u32gTotalDistanceRawValue := TO_UDINT((u32gTotalDistance.Value - u32gTotalDistance.AppScalingOffset) * u32gTotalDistance.AppScalingDivisor / u32gTotalDistance.AppScalingMultiplier);

                  
END_GET
END_PROPERTY

PROPERTY i32gDistanceTraveledMeasureMastToolValue : DINT
GET
                    IF i32gDistanceTraveledMeasureMast.ToolScalingDivisor = 0 OR i32gDistanceTraveledMeasureMast.AppScalingMultiplier = 0 THEN
	_MatchLog^.Error("Get i32gDistanceTraveledMeasureMastToolValue", "Division by Zero!");
	RETURN;
END_IF

i32gDistanceTraveledMeasureMastToolValue := TO_DINT(((i32gDistanceTraveledMeasureMast.Value - i32gDistanceTraveledMeasureMast.AppScalingOffset) * i32gDistanceTraveledMeasureMast.AppScalingDivisor / i32gDistanceTraveledMeasureMast.AppScalingMultiplier * i32gDistanceTraveledMeasureMast.ToolScalingMultiplier / i32gDistanceTraveledMeasureMast.ToolScalingDivisor) + i32gDistanceTraveledMeasureMast.ToolScalingOffset);

                  
END_GET
END_PROPERTY

PROPERTY u32gTotalDistanceToolValue : UDINT
GET
                    IF u32gTotalDistance.ToolScalingDivisor = 0 OR u32gTotalDistance.AppScalingMultiplier = 0 THEN
	_MatchLog^.Error("Get u32gTotalDistanceToolValue", "Division by Zero!");
	RETURN;
END_IF

u32gTotalDistanceToolValue := TO_UDINT(((u32gTotalDistance.Value - u32gTotalDistance.AppScalingOffset) * u32gTotalDistance.AppScalingDivisor / u32gTotalDistance.AppScalingMultiplier * u32gTotalDistance.ToolScalingMultiplier / u32gTotalDistance.ToolScalingDivisor) + u32gTotalDistance.ToolScalingOffset);

                  
END_GET
END_PROPERTY

METHOD InitializeCanSignals
                  i32gDistanceTraveledMeasureMast.AppScalingDivisor :=1;
i32gDistanceTraveledMeasureMast.AppScalingMultiplier :=1;
i32gDistanceTraveledMeasureMast.AppScalingOffset :=0;
i32gDistanceTraveledMeasureMast.AppUnit :="";
i32gDistanceTraveledMeasureMast.CanDefault :=0;
i32gDistanceTraveledMeasureMast.CanInit :=0;
i32gDistanceTraveledMeasureMast.CanMax :=VBasic.LibConst.I32_MAX;
i32gDistanceTraveledMeasureMast.CanMin :=VBasic.LibConst.32_MIN;
i32gDistanceTraveledMeasureMast.CanUnit :="";
i32gDistanceTraveledMeasureMast.Description :="new signal";
i32gDistanceTraveledMeasureMast.ErrorReaction := eErrorReaction.ERSIG_DFLT;
i32gDistanceTraveledMeasureMast.ReceiverAdress :=1;
i32gDistanceTraveledMeasureMast.ToolScalingDivisor :=1;
i32gDistanceTraveledMeasureMast.ToolScalingMultiplier :=1;
i32gDistanceTraveledMeasureMast.ToolScalingOffset :=0;
i32gDistanceTraveledMeasureMast.ToolUnit :="";

u32gTotalDistance.AppScalingDivisor :=1;
u32gTotalDistance.AppScalingMultiplier :=1;
u32gTotalDistance.AppScalingOffset :=0;
u32gTotalDistance.AppUnit :="";
u32gTotalDistance.CanDefault :=0;
u32gTotalDistance.CanInit :=0;
u32gTotalDistance.CanMax :=VBasic.LibConst.U32_MAX;
u32gTotalDistance.CanMin :=VBasic.LibConst.U32_MIN;
u32gTotalDistance.CanUnit :="";
u32gTotalDistance.Description :="new signal";
u32gTotalDistance.ErrorReaction := eErrorReaction.ERSIG_DFLT;
u32gTotalDistance.ReceiverAdress :=1;
u32gTotalDistance.ToolScalingDivisor :=1;
u32gTotalDistance.ToolScalingMultiplier :=1;
u32gTotalDistance.ToolScalingOffset :=0;
u32gTotalDistance.ToolUnit :="";


                
END_METHOD
END_FUNCTION_BLOCK

FUNCTION_BLOCK Msg13C0SendToEvision7MessageClass EXTENDS CanReceiveMessageClass
  VAR_INPUT
    u8gReductionPumpRail : UInt8CanSignalClass;
    u8gPourcentCycleBrake : UInt8CanSignalClass;
    u8gPourcentCycle2ndParkBrake : UInt8CanSignalClass;
    bogSecondParkBrakeActive : BoolCanSignalClass;
    boStatFront2eParkTrainBrakeTest : BoolCanSignalClass;
    boStatBack2eParkTrainBrakeTest : BoolCanSignalClass;
    boAutorizeRazController : BoolCanSignalClass;
    boVoltageDcConverterFault : BoolCanSignalClass;
    boBatteryLowLevel : BoolCanSignalClass;
    boBattErrorCode1 : BoolCanSignalClass;
    boActiveFaultRazDmc : BoolCanSignalClass;
    i16Motor_Rpm : Int16CanSignalClass;
    i8Controller_Temp : Int8CanSignalClass;
    i8Motor_Temp : Int8CanSignalClass;
    Counter : UInt32CanSignalClass;
  END_VAR

            
          

METHOD SetData
  VAR_INPUT
    CanMsgPointer : POINTER TO CanMessageClass;
  END_VAR
                  IF IsValidPointer(canMsgPointer,'SetData') THEN
	SUPER^.SetData(CanMsgPointer);
	//Set the new data
	u8gReductionPumpRail.Value := canMsgPointer^.GetUint8(0);
	u8gPourcentCycleBrake.Value := canMsgPointer^.GetUint8(8);
	u8gPourcentCycle2ndParkBrake.Value := canMsgPointer^.GetUint8(16);
	bogSecondParkBrakeActive.Value := canMsgPointer^.GetBoolOnBit(24);
	boStatFront2eParkTrainBrakeTest.Value := canMsgPointer^.GetBoolOnBit(25);
	boStatBack2eParkTrainBrakeTest.Value := canMsgPointer^.GetBoolOnBit(26);
	boAutorizeRazController.Value := canMsgPointer^.GetBoolOnBit(27);
	boVoltageDcConverterFault.Value := canMsgPointer^.GetBoolOnBit(28);
	boBatteryLowLevel.Value := canMsgPointer^.GetBoolOnBit(29);
	boBattErrorCode1.Value := canMsgPointer^.GetBoolOnBit(30);
	boActiveFaultRazDmc.Value := canMsgPointer^.GetBoolOnBit(31);
	i16Motor_Rpm.Value := canMsgPointer^.GetInt16(32);
	i8Controller_Temp.Value := canMsgPointer^.GetInt8(48);
	i8Motor_Temp.Value := canMsgPointer^.GetInt8(56);
	//And increase the counter
	Counter.Value := CanMsgPointer^.Counter.Value;
END_IF

                
END_METHOD

PROPERTY u8gReductionPumpRailRawValue : USINT
GET
                    IF u8gReductionPumpRail.AppScalingMultiplier = 0 THEN
	_MatchLog^.Error("Get u8gReductionPumpRailRawValue", "Division by Zero!");
	RETURN;
End_IF

u8gReductionPumpRailRawValue := TO_USINT((u8gReductionPumpRail.Value - u8gReductionPumpRail.AppScalingOffset) * u8gReductionPumpRail.AppScalingDivisor / u8gReductionPumpRail.AppScalingMultiplier);

                  
END_GET
END_PROPERTY

PROPERTY u8gPourcentCycleBrakeRawValue : USINT
GET
                    IF u8gPourcentCycleBrake.AppScalingMultiplier = 0 THEN
	_MatchLog^.Error("Get u8gPourcentCycleBrakeRawValue", "Division by Zero!");
	RETURN;
End_IF

u8gPourcentCycleBrakeRawValue := TO_USINT((u8gPourcentCycleBrake.Value - u8gPourcentCycleBrake.AppScalingOffset) * u8gPourcentCycleBrake.AppScalingDivisor / u8gPourcentCycleBrake.AppScalingMultiplier);

                  
END_GET
END_PROPERTY

PROPERTY u8gPourcentCycle2ndParkBrakeRawValue : USINT
GET
                    IF u8gPourcentCycle2ndParkBrake.AppScalingMultiplier = 0 THEN
	_MatchLog^.Error("Get u8gPourcentCycle2ndParkBrakeRawValue", "Division by Zero!");
	RETURN;
End_IF

u8gPourcentCycle2ndParkBrakeRawValue := TO_USINT((u8gPourcentCycle2ndParkBrake.Value - u8gPourcentCycle2ndParkBrake.AppScalingOffset) * u8gPourcentCycle2ndParkBrake.AppScalingDivisor / u8gPourcentCycle2ndParkBrake.AppScalingMultiplier);

                  
END_GET
END_PROPERTY

PROPERTY bogSecondParkBrakeActiveRawValue : BOOL
GET
                    bogSecondParkBrakeActiveRawValue := bogSecondParkBrakeActive.Value;

                  
END_GET
END_PROPERTY

PROPERTY boStatFront2eParkTrainBrakeTestRawValue : BOOL
GET
                    boStatFront2eParkTrainBrakeTestRawValue := boStatFront2eParkTrainBrakeTest.Value;

                  
END_GET
END_PROPERTY

PROPERTY boStatBack2eParkTrainBrakeTestRawValue : BOOL
GET
                    boStatBack2eParkTrainBrakeTestRawValue := boStatBack2eParkTrainBrakeTest.Value;

                  
END_GET
END_PROPERTY

PROPERTY boAutorizeRazControllerRawValue : BOOL
GET
                    boAutorizeRazControllerRawValue := boAutorizeRazController.Value;

                  
END_GET
END_PROPERTY

PROPERTY boVoltageDcConverterFaultRawValue : BOOL
GET
                    boVoltageDcConverterFaultRawValue := boVoltageDcConverterFault.Value;

                  
END_GET
END_PROPERTY

PROPERTY boBatteryLowLevelRawValue : BOOL
GET
                    boBatteryLowLevelRawValue := boBatteryLowLevel.Value;

                  
END_GET
END_PROPERTY

PROPERTY boBattErrorCode1RawValue : BOOL
GET
                    boBattErrorCode1RawValue := boBattErrorCode1.Value;

                  
END_GET
END_PROPERTY

PROPERTY boActiveFaultRazDmcRawValue : BOOL
GET
                    boActiveFaultRazDmcRawValue := boActiveFaultRazDmc.Value;

                  
END_GET
END_PROPERTY

PROPERTY i16Motor_RpmRawValue : INT
GET
                    IF i16Motor_Rpm.AppScalingMultiplier = 0 THEN
	_MatchLog^.Error("Get i16Motor_RpmRawValue", "Division by Zero!");
	RETURN;
End_IF

i16Motor_RpmRawValue := TO_INT((i16Motor_Rpm.Value - i16Motor_Rpm.AppScalingOffset) * i16Motor_Rpm.AppScalingDivisor / i16Motor_Rpm.AppScalingMultiplier);

                  
END_GET
END_PROPERTY

PROPERTY i8Controller_TempRawValue : SINT
GET
                    IF i8Controller_Temp.AppScalingMultiplier = 0 THEN
	_MatchLog^.Error("Get i8Controller_TempRawValue", "Division by Zero!");
	RETURN;
End_IF

i8Controller_TempRawValue := TO_SINT((i8Controller_Temp.Value - i8Controller_Temp.AppScalingOffset) * i8Controller_Temp.AppScalingDivisor / i8Controller_Temp.AppScalingMultiplier);

                  
END_GET
END_PROPERTY

PROPERTY i8Motor_TempRawValue : SINT
GET
                    IF i8Motor_Temp.AppScalingMultiplier = 0 THEN
	_MatchLog^.Error("Get i8Motor_TempRawValue", "Division by Zero!");
	RETURN;
End_IF

i8Motor_TempRawValue := TO_SINT((i8Motor_Temp.Value - i8Motor_Temp.AppScalingOffset) * i8Motor_Temp.AppScalingDivisor / i8Motor_Temp.AppScalingMultiplier);

                  
END_GET
END_PROPERTY

PROPERTY u8gReductionPumpRailToolValue : USINT
GET
                    IF u8gReductionPumpRail.ToolScalingDivisor = 0 OR u8gReductionPumpRail.AppScalingMultiplier = 0 THEN
	_MatchLog^.Error("Get u8gReductionPumpRailToolValue", "Division by Zero!");
	RETURN;
END_IF

u8gReductionPumpRailToolValue := TO_USINT(((u8gReductionPumpRail.Value - u8gReductionPumpRail.AppScalingOffset) * u8gReductionPumpRail.AppScalingDivisor / u8gReductionPumpRail.AppScalingMultiplier * u8gReductionPumpRail.ToolScalingMultiplier / u8gReductionPumpRail.ToolScalingDivisor) + u8gReductionPumpRail.ToolScalingOffset);

                  
END_GET
END_PROPERTY

PROPERTY u8gPourcentCycleBrakeToolValue : USINT
GET
                    IF u8gPourcentCycleBrake.ToolScalingDivisor = 0 OR u8gPourcentCycleBrake.AppScalingMultiplier = 0 THEN
	_MatchLog^.Error("Get u8gPourcentCycleBrakeToolValue", "Division by Zero!");
	RETURN;
END_IF

u8gPourcentCycleBrakeToolValue := TO_USINT(((u8gPourcentCycleBrake.Value - u8gPourcentCycleBrake.AppScalingOffset) * u8gPourcentCycleBrake.AppScalingDivisor / u8gPourcentCycleBrake.AppScalingMultiplier * u8gPourcentCycleBrake.ToolScalingMultiplier / u8gPourcentCycleBrake.ToolScalingDivisor) + u8gPourcentCycleBrake.ToolScalingOffset);

                  
END_GET
END_PROPERTY

PROPERTY u8gPourcentCycle2ndParkBrakeToolValue : USINT
GET
                    IF u8gPourcentCycle2ndParkBrake.ToolScalingDivisor = 0 OR u8gPourcentCycle2ndParkBrake.AppScalingMultiplier = 0 THEN
	_MatchLog^.Error("Get u8gPourcentCycle2ndParkBrakeToolValue", "Division by Zero!");
	RETURN;
END_IF

u8gPourcentCycle2ndParkBrakeToolValue := TO_USINT(((u8gPourcentCycle2ndParkBrake.Value - u8gPourcentCycle2ndParkBrake.AppScalingOffset) * u8gPourcentCycle2ndParkBrake.AppScalingDivisor / u8gPourcentCycle2ndParkBrake.AppScalingMultiplier * u8gPourcentCycle2ndParkBrake.ToolScalingMultiplier / u8gPourcentCycle2ndParkBrake.ToolScalingDivisor) + u8gPourcentCycle2ndParkBrake.ToolScalingOffset);

                  
END_GET
END_PROPERTY

PROPERTY bogSecondParkBrakeActiveToolValue : BOOL
GET
                    bogSecondParkBrakeActiveToolValue := bogSecondParkBrakeActive.Value;

                  
END_GET
END_PROPERTY

PROPERTY boStatFront2eParkTrainBrakeTestToolValue : BOOL
GET
                    boStatFront2eParkTrainBrakeTestToolValue := boStatFront2eParkTrainBrakeTest.Value;

                  
END_GET
END_PROPERTY

PROPERTY boStatBack2eParkTrainBrakeTestToolValue : BOOL
GET
                    boStatBack2eParkTrainBrakeTestToolValue := boStatBack2eParkTrainBrakeTest.Value;

                  
END_GET
END_PROPERTY

PROPERTY boAutorizeRazControllerToolValue : BOOL
GET
                    boAutorizeRazControllerToolValue := boAutorizeRazController.Value;

                  
END_GET
END_PROPERTY

PROPERTY boVoltageDcConverterFaultToolValue : BOOL
GET
                    boVoltageDcConverterFaultToolValue := boVoltageDcConverterFault.Value;

                  
END_GET
END_PROPERTY

PROPERTY boBatteryLowLevelToolValue : BOOL
GET
                    boBatteryLowLevelToolValue := boBatteryLowLevel.Value;

                  
END_GET
END_PROPERTY

PROPERTY boBattErrorCode1ToolValue : BOOL
GET
                    boBattErrorCode1ToolValue := boBattErrorCode1.Value;

                  
END_GET
END_PROPERTY

PROPERTY boActiveFaultRazDmcToolValue : BOOL
GET
                    boActiveFaultRazDmcToolValue := boActiveFaultRazDmc.Value;

                  
END_GET
END_PROPERTY

PROPERTY i16Motor_RpmToolValue : INT
GET
                    IF i16Motor_Rpm.ToolScalingDivisor = 0 OR i16Motor_Rpm.AppScalingMultiplier = 0 THEN
	_MatchLog^.Error("Get i16Motor_RpmToolValue", "Division by Zero!");
	RETURN;
END_IF

i16Motor_RpmToolValue := TO_INT(((i16Motor_Rpm.Value - i16Motor_Rpm.AppScalingOffset) * i16Motor_Rpm.AppScalingDivisor / i16Motor_Rpm.AppScalingMultiplier * i16Motor_Rpm.ToolScalingMultiplier / i16Motor_Rpm.ToolScalingDivisor) + i16Motor_Rpm.ToolScalingOffset);

                  
END_GET
END_PROPERTY

PROPERTY i8Controller_TempToolValue : SINT
GET
                    IF i8Controller_Temp.ToolScalingDivisor = 0 OR i8Controller_Temp.AppScalingMultiplier = 0 THEN
	_MatchLog^.Error("Get i8Controller_TempToolValue", "Division by Zero!");
	RETURN;
END_IF

i8Controller_TempToolValue := TO_SINT(((i8Controller_Temp.Value - i8Controller_Temp.AppScalingOffset) * i8Controller_Temp.AppScalingDivisor / i8Controller_Temp.AppScalingMultiplier * i8Controller_Temp.ToolScalingMultiplier / i8Controller_Temp.ToolScalingDivisor) + i8Controller_Temp.ToolScalingOffset);

                  
END_GET
END_PROPERTY

PROPERTY i8Motor_TempToolValue : SINT
GET
                    IF i8Motor_Temp.ToolScalingDivisor = 0 OR i8Motor_Temp.AppScalingMultiplier = 0 THEN
	_MatchLog^.Error("Get i8Motor_TempToolValue", "Division by Zero!");
	RETURN;
END_IF

i8Motor_TempToolValue := TO_SINT(((i8Motor_Temp.Value - i8Motor_Temp.AppScalingOffset) * i8Motor_Temp.AppScalingDivisor / i8Motor_Temp.AppScalingMultiplier * i8Motor_Temp.ToolScalingMultiplier / i8Motor_Temp.ToolScalingDivisor) + i8Motor_Temp.ToolScalingOffset);

                  
END_GET
END_PROPERTY

METHOD InitializeCanSignals
                  u8gReductionPumpRail.AppScalingDivisor :=1;
u8gReductionPumpRail.AppScalingMultiplier :=1;
u8gReductionPumpRail.AppScalingOffset :=0;
u8gReductionPumpRail.AppUnit :="";
u8gReductionPumpRail.CanDefault :=0;
u8gReductionPumpRail.CanInit :=0;
u8gReductionPumpRail.CanMax :=VBasic.LibConst.U8_MAX;
u8gReductionPumpRail.CanMin :=VBasic.LibConst.U8_MIN;
u8gReductionPumpRail.CanUnit :="";
u8gReductionPumpRail.Description :="new signal";
u8gReductionPumpRail.ErrorReaction := eErrorReaction.ERSIG_DFLT;
u8gReductionPumpRail.ReceiverAdress :=1;
u8gReductionPumpRail.ToolScalingDivisor :=1;
u8gReductionPumpRail.ToolScalingMultiplier :=1;
u8gReductionPumpRail.ToolScalingOffset :=0;
u8gReductionPumpRail.ToolUnit :="";

u8gPourcentCycleBrake.AppScalingDivisor :=1;
u8gPourcentCycleBrake.AppScalingMultiplier :=1;
u8gPourcentCycleBrake.AppScalingOffset :=0;
u8gPourcentCycleBrake.AppUnit :="";
u8gPourcentCycleBrake.CanDefault :=0;
u8gPourcentCycleBrake.CanInit :=0;
u8gPourcentCycleBrake.CanMax :=VBasic.LibConst.U8_MAX;
u8gPourcentCycleBrake.CanMin :=VBasic.LibConst.U8_MIN;
u8gPourcentCycleBrake.CanUnit :="";
u8gPourcentCycleBrake.Description :="new signal";
u8gPourcentCycleBrake.ErrorReaction := eErrorReaction.ERSIG_DFLT;
u8gPourcentCycleBrake.ReceiverAdress :=1;
u8gPourcentCycleBrake.ToolScalingDivisor :=1;
u8gPourcentCycleBrake.ToolScalingMultiplier :=1;
u8gPourcentCycleBrake.ToolScalingOffset :=0;
u8gPourcentCycleBrake.ToolUnit :="";

u8gPourcentCycle2ndParkBrake.AppScalingDivisor :=1;
u8gPourcentCycle2ndParkBrake.AppScalingMultiplier :=1;
u8gPourcentCycle2ndParkBrake.AppScalingOffset :=0;
u8gPourcentCycle2ndParkBrake.AppUnit :="";
u8gPourcentCycle2ndParkBrake.CanDefault :=0;
u8gPourcentCycle2ndParkBrake.CanInit :=0;
u8gPourcentCycle2ndParkBrake.CanMax :=VBasic.LibConst.U8_MAX;
u8gPourcentCycle2ndParkBrake.CanMin :=VBasic.LibConst.U8_MIN;
u8gPourcentCycle2ndParkBrake.CanUnit :="";
u8gPourcentCycle2ndParkBrake.Description :="Envoie du pourcentage du nombre de cycle de freins";
u8gPourcentCycle2ndParkBrake.ErrorReaction := eErrorReaction.ERSIG_DFLT;
u8gPourcentCycle2ndParkBrake.ReceiverAdress :=1;
u8gPourcentCycle2ndParkBrake.ToolScalingDivisor :=1;
u8gPourcentCycle2ndParkBrake.ToolScalingMultiplier :=1;
u8gPourcentCycle2ndParkBrake.ToolScalingOffset :=0;
u8gPourcentCycle2ndParkBrake.ToolUnit :="";

bogSecondParkBrakeActive.AppScalingDivisor :=1;
bogSecondParkBrakeActive.AppScalingMultiplier :=1;
bogSecondParkBrakeActive.AppScalingOffset :=0;
bogSecondParkBrakeActive.AppUnit :="";
bogSecondParkBrakeActive.CanDefault :=0;
bogSecondParkBrakeActive.CanInit :=0;
bogSecondParkBrakeActive.CanMax :=1;
bogSecondParkBrakeActive.CanMin :=0;
bogSecondParkBrakeActive.CanUnit :="";
bogSecondParkBrakeActive.Description :="Option active";
bogSecondParkBrakeActive.ErrorReaction := eErrorReaction.ERSIG_DFLT;
bogSecondParkBrakeActive.ReceiverAdress :=1;
bogSecondParkBrakeActive.ToolScalingDivisor :=1;
bogSecondParkBrakeActive.ToolScalingMultiplier :=1;
bogSecondParkBrakeActive.ToolScalingOffset :=0;
bogSecondParkBrakeActive.ToolUnit :="";

boStatFront2eParkTrainBrakeTest.AppScalingDivisor :=1;
boStatFront2eParkTrainBrakeTest.AppScalingMultiplier :=1;
boStatFront2eParkTrainBrakeTest.AppScalingOffset :=0;
boStatFront2eParkTrainBrakeTest.AppUnit :="";
boStatFront2eParkTrainBrakeTest.CanDefault :=0;
boStatFront2eParkTrainBrakeTest.CanInit :=0;
boStatFront2eParkTrainBrakeTest.CanMax :=1;
boStatFront2eParkTrainBrakeTest.CanMin :=0;
boStatFront2eParkTrainBrakeTest.CanUnit :="";
boStatFront2eParkTrainBrakeTest.Description :="Validation du test frein sur le 2nd frein de oscillant";
boStatFront2eParkTrainBrakeTest.ErrorReaction := eErrorReaction.ERSIG_DFLT;
boStatFront2eParkTrainBrakeTest.ReceiverAdress :=1;
boStatFront2eParkTrainBrakeTest.ToolScalingDivisor :=1;
boStatFront2eParkTrainBrakeTest.ToolScalingMultiplier :=1;
boStatFront2eParkTrainBrakeTest.ToolScalingOffset :=0;
boStatFront2eParkTrainBrakeTest.ToolUnit :="";

boStatBack2eParkTrainBrakeTest.AppScalingDivisor :=1;
boStatBack2eParkTrainBrakeTest.AppScalingMultiplier :=1;
boStatBack2eParkTrainBrakeTest.AppScalingOffset :=0;
boStatBack2eParkTrainBrakeTest.AppUnit :="";
boStatBack2eParkTrainBrakeTest.CanDefault :=0;
boStatBack2eParkTrainBrakeTest.CanInit :=0;
boStatBack2eParkTrainBrakeTest.CanMax :=1;
boStatBack2eParkTrainBrakeTest.CanMin :=0;
boStatBack2eParkTrainBrakeTest.CanUnit :="";
boStatBack2eParkTrainBrakeTest.Description :="Validation du test frein sur le 2nd frein du fixe";
boStatBack2eParkTrainBrakeTest.ErrorReaction := eErrorReaction.ERSIG_DFLT;
boStatBack2eParkTrainBrakeTest.ReceiverAdress :=1;
boStatBack2eParkTrainBrakeTest.ToolScalingDivisor :=1;
boStatBack2eParkTrainBrakeTest.ToolScalingMultiplier :=1;
boStatBack2eParkTrainBrakeTest.ToolScalingOffset :=0;
boStatBack2eParkTrainBrakeTest.ToolUnit :="";

boAutorizeRazController.AppScalingDivisor :=1;
boAutorizeRazController.AppScalingMultiplier :=1;
boAutorizeRazController.AppScalingOffset :=0;
boAutorizeRazController.AppUnit :="";
boAutorizeRazController.CanDefault :=0;
boAutorizeRazController.CanInit :=0;
boAutorizeRazController.CanMax :=1;
boAutorizeRazController.CanMin :=0;
boAutorizeRazController.CanUnit :="";
boAutorizeRazController.Description :="new signal";
boAutorizeRazController.ErrorReaction := eErrorReaction.ERSIG_DFLT;
boAutorizeRazController.ReceiverAdress :=1;
boAutorizeRazController.ToolScalingDivisor :=1;
boAutorizeRazController.ToolScalingMultiplier :=1;
boAutorizeRazController.ToolScalingOffset :=0;
boAutorizeRazController.ToolUnit :="";

boVoltageDcConverterFault.AppScalingDivisor :=1;
boVoltageDcConverterFault.AppScalingMultiplier :=1;
boVoltageDcConverterFault.AppScalingOffset :=0;
boVoltageDcConverterFault.AppUnit :="";
boVoltageDcConverterFault.CanDefault :=0;
boVoltageDcConverterFault.CanInit :=0;
boVoltageDcConverterFault.CanMax :=1;
boVoltageDcConverterFault.CanMin :=0;
boVoltageDcConverterFault.CanUnit :="";
boVoltageDcConverterFault.Description :="new signal";
boVoltageDcConverterFault.ErrorReaction := eErrorReaction.ERSIG_DFLT;
boVoltageDcConverterFault.ReceiverAdress :=1;
boVoltageDcConverterFault.ToolScalingDivisor :=1;
boVoltageDcConverterFault.ToolScalingMultiplier :=1;
boVoltageDcConverterFault.ToolScalingOffset :=0;
boVoltageDcConverterFault.ToolUnit :="";

boBatteryLowLevel.AppScalingDivisor :=1;
boBatteryLowLevel.AppScalingMultiplier :=1;
boBatteryLowLevel.AppScalingOffset :=0;
boBatteryLowLevel.AppUnit :="";
boBatteryLowLevel.CanDefault :=0;
boBatteryLowLevel.CanInit :=0;
boBatteryLowLevel.CanMax :=1;
boBatteryLowLevel.CanMin :=0;
boBatteryLowLevel.CanUnit :="";
boBatteryLowLevel.Description :="new signal";
boBatteryLowLevel.ErrorReaction := eErrorReaction.ERSIG_DFLT;
boBatteryLowLevel.ReceiverAdress :=1;
boBatteryLowLevel.ToolScalingDivisor :=1;
boBatteryLowLevel.ToolScalingMultiplier :=1;
boBatteryLowLevel.ToolScalingOffset :=0;
boBatteryLowLevel.ToolUnit :="";

boBattErrorCode1.AppScalingDivisor :=1;
boBattErrorCode1.AppScalingMultiplier :=1;
boBattErrorCode1.AppScalingOffset :=0;
boBattErrorCode1.AppUnit :="";
boBattErrorCode1.CanDefault :=0;
boBattErrorCode1.CanInit :=0;
boBattErrorCode1.CanMax :=1;
boBattErrorCode1.CanMin :=0;
boBattErrorCode1.CanUnit :="";
boBattErrorCode1.Description :="new signal";
boBattErrorCode1.ErrorReaction := eErrorReaction.ERSIG_DFLT;
boBattErrorCode1.ReceiverAdress :=1;
boBattErrorCode1.ToolScalingDivisor :=1;
boBattErrorCode1.ToolScalingMultiplier :=1;
boBattErrorCode1.ToolScalingOffset :=0;
boBattErrorCode1.ToolUnit :="";

boActiveFaultRazDmc.AppScalingDivisor :=1;
boActiveFaultRazDmc.AppScalingMultiplier :=1;
boActiveFaultRazDmc.AppScalingOffset :=0;
boActiveFaultRazDmc.AppUnit :="";
boActiveFaultRazDmc.CanDefault :=0;
boActiveFaultRazDmc.CanInit :=0;
boActiveFaultRazDmc.CanMax :=1;
boActiveFaultRazDmc.CanMin :=0;
boActiveFaultRazDmc.CanUnit :="";
boActiveFaultRazDmc.Description :="new signal";
boActiveFaultRazDmc.ErrorReaction := eErrorReaction.ERSIG_DFLT;
boActiveFaultRazDmc.ReceiverAdress :=1;
boActiveFaultRazDmc.ToolScalingDivisor :=1;
boActiveFaultRazDmc.ToolScalingMultiplier :=1;
boActiveFaultRazDmc.ToolScalingOffset :=0;
boActiveFaultRazDmc.ToolUnit :="";

i16Motor_Rpm.AppScalingDivisor :=1;
i16Motor_Rpm.AppScalingMultiplier :=1;
i16Motor_Rpm.AppScalingOffset :=0;
i16Motor_Rpm.AppUnit :="";
i16Motor_Rpm.CanDefault :=0;
i16Motor_Rpm.CanInit :=0;
i16Motor_Rpm.CanMax :=VBasic.LibConst.I16_MAX;
i16Motor_Rpm.CanMin :=VBasic.LibConst.I16_MIN;
i16Motor_Rpm.CanUnit :="";
i16Motor_Rpm.Description :="new signal";
i16Motor_Rpm.ErrorReaction := eErrorReaction.ERSIG_DFLT;
i16Motor_Rpm.ReceiverAdress :=1;
i16Motor_Rpm.ToolScalingDivisor :=1;
i16Motor_Rpm.ToolScalingMultiplier :=1;
i16Motor_Rpm.ToolScalingOffset :=0;
i16Motor_Rpm.ToolUnit :="";

i8Controller_Temp.AppScalingDivisor :=1;
i8Controller_Temp.AppScalingMultiplier :=1;
i8Controller_Temp.AppScalingOffset :=0;
i8Controller_Temp.AppUnit :="";
i8Controller_Temp.CanDefault :=0;
i8Controller_Temp.CanInit :=0;
i8Controller_Temp.CanMax :=VBasic.LibConst.I8_MAX;
i8Controller_Temp.CanMin :=VBasic.LibConst.I8_MIN;
i8Controller_Temp.CanUnit :="";
i8Controller_Temp.Description :="new signal";
i8Controller_Temp.ErrorReaction := eErrorReaction.ERSIG_DFLT;
i8Controller_Temp.ReceiverAdress :=1;
i8Controller_Temp.ToolScalingDivisor :=1;
i8Controller_Temp.ToolScalingMultiplier :=1;
i8Controller_Temp.ToolScalingOffset :=0;
i8Controller_Temp.ToolUnit :="";

i8Motor_Temp.AppScalingDivisor :=1;
i8Motor_Temp.AppScalingMultiplier :=1;
i8Motor_Temp.AppScalingOffset :=0;
i8Motor_Temp.AppUnit :="";
i8Motor_Temp.CanDefault :=0;
i8Motor_Temp.CanInit :=0;
i8Motor_Temp.CanMax :=VBasic.LibConst.I8_MAX;
i8Motor_Temp.CanMin :=VBasic.LibConst.I8_MIN;
i8Motor_Temp.CanUnit :="";
i8Motor_Temp.Description :="new signal";
i8Motor_Temp.ErrorReaction := eErrorReaction.ERSIG_DFLT;
i8Motor_Temp.ReceiverAdress :=1;
i8Motor_Temp.ToolScalingDivisor :=1;
i8Motor_Temp.ToolScalingMultiplier :=1;
i8Motor_Temp.ToolScalingOffset :=0;
i8Motor_Temp.ToolUnit :="";


                
END_METHOD
END_FUNCTION_BLOCK

FUNCTION_BLOCK Msg14C0SendToEvision7MessageClass EXTENDS CanReceiveMessageClass
  VAR_INPUT
    i16Ibatt_ist : Int16CanSignalClass;
    u16Vbatt_ist : UInt16CanSignalClass;
    u8Batt_Soc : UInt8CanSignalClass;
    boAddParkBrakeActive : BoolCanSignalClass;
    boPreventLimitSpeedExceeding : BoolCanSignalClass;
    Counter : UInt32CanSignalClass;
  END_VAR

            
          

METHOD SetData
  VAR_INPUT
    CanMsgPointer : POINTER TO CanMessageClass;
  END_VAR
                  IF IsValidPointer(canMsgPointer,'SetData') THEN
	SUPER^.SetData(CanMsgPointer);
	//Set the new data
	i16Ibatt_ist.Value := canMsgPointer^.GetInt16(0);
	u16Vbatt_ist.Value := canMsgPointer^.GetUint16(16);
	u8Batt_Soc.Value := canMsgPointer^.GetUint8(32);
	boAddParkBrakeActive.Value := canMsgPointer^.GetBoolOnBit(56);
	boPreventLimitSpeedExceeding.Value := canMsgPointer^.GetBoolOnBit(57);
	//And increase the counter
	Counter.Value := CanMsgPointer^.Counter.Value;
END_IF

                
END_METHOD

PROPERTY i16Ibatt_istRawValue : INT
GET
                    IF i16Ibatt_ist.AppScalingMultiplier = 0 THEN
	_MatchLog^.Error("Get i16Ibatt_istRawValue", "Division by Zero!");
	RETURN;
End_IF

i16Ibatt_istRawValue := TO_INT((i16Ibatt_ist.Value - i16Ibatt_ist.AppScalingOffset) * i16Ibatt_ist.AppScalingDivisor / i16Ibatt_ist.AppScalingMultiplier);

                  
END_GET
END_PROPERTY

PROPERTY u16Vbatt_istRawValue : UINT
GET
                    IF u16Vbatt_ist.AppScalingMultiplier = 0 THEN
	_MatchLog^.Error("Get u16Vbatt_istRawValue", "Division by Zero!");
	RETURN;
End_IF

u16Vbatt_istRawValue := TO_UINT((u16Vbatt_ist.Value - u16Vbatt_ist.AppScalingOffset) * u16Vbatt_ist.AppScalingDivisor / u16Vbatt_ist.AppScalingMultiplier);

                  
END_GET
END_PROPERTY

PROPERTY u8Batt_SocRawValue : USINT
GET
                    IF u8Batt_Soc.AppScalingMultiplier = 0 THEN
	_MatchLog^.Error("Get u8Batt_SocRawValue", "Division by Zero!");
	RETURN;
End_IF

u8Batt_SocRawValue := TO_USINT((u8Batt_Soc.Value - u8Batt_Soc.AppScalingOffset) * u8Batt_Soc.AppScalingDivisor / u8Batt_Soc.AppScalingMultiplier);

                  
END_GET
END_PROPERTY

PROPERTY boAddParkBrakeActiveRawValue : BOOL
GET
                    boAddParkBrakeActiveRawValue := boAddParkBrakeActive.Value;

                  
END_GET
END_PROPERTY

PROPERTY boPreventLimitSpeedExceedingRawValue : BOOL
GET
                    boPreventLimitSpeedExceedingRawValue := boPreventLimitSpeedExceeding.Value;

                  
END_GET
END_PROPERTY

PROPERTY i16Ibatt_istToolValue : INT
GET
                    IF i16Ibatt_ist.ToolScalingDivisor = 0 OR i16Ibatt_ist.AppScalingMultiplier = 0 THEN
	_MatchLog^.Error("Get i16Ibatt_istToolValue", "Division by Zero!");
	RETURN;
END_IF

i16Ibatt_istToolValue := TO_INT(((i16Ibatt_ist.Value - i16Ibatt_ist.AppScalingOffset) * i16Ibatt_ist.AppScalingDivisor / i16Ibatt_ist.AppScalingMultiplier * i16Ibatt_ist.ToolScalingMultiplier / i16Ibatt_ist.ToolScalingDivisor) + i16Ibatt_ist.ToolScalingOffset);

                  
END_GET
END_PROPERTY

PROPERTY u16Vbatt_istToolValue : UINT
GET
                    IF u16Vbatt_ist.ToolScalingDivisor = 0 OR u16Vbatt_ist.AppScalingMultiplier = 0 THEN
	_MatchLog^.Error("Get u16Vbatt_istToolValue", "Division by Zero!");
	RETURN;
END_IF

u16Vbatt_istToolValue := TO_UINT(((u16Vbatt_ist.Value - u16Vbatt_ist.AppScalingOffset) * u16Vbatt_ist.AppScalingDivisor / u16Vbatt_ist.AppScalingMultiplier * u16Vbatt_ist.ToolScalingMultiplier / u16Vbatt_ist.ToolScalingDivisor) + u16Vbatt_ist.ToolScalingOffset);

                  
END_GET
END_PROPERTY

PROPERTY u8Batt_SocToolValue : USINT
GET
                    IF u8Batt_Soc.ToolScalingDivisor = 0 OR u8Batt_Soc.AppScalingMultiplier = 0 THEN
	_MatchLog^.Error("Get u8Batt_SocToolValue", "Division by Zero!");
	RETURN;
END_IF

u8Batt_SocToolValue := TO_USINT(((u8Batt_Soc.Value - u8Batt_Soc.AppScalingOffset) * u8Batt_Soc.AppScalingDivisor / u8Batt_Soc.AppScalingMultiplier * u8Batt_Soc.ToolScalingMultiplier / u8Batt_Soc.ToolScalingDivisor) + u8Batt_Soc.ToolScalingOffset);

                  
END_GET
END_PROPERTY

PROPERTY boAddParkBrakeActiveToolValue : BOOL
GET
                    boAddParkBrakeActiveToolValue := boAddParkBrakeActive.Value;

                  
END_GET
END_PROPERTY

PROPERTY boPreventLimitSpeedExceedingToolValue : BOOL
GET
                    boPreventLimitSpeedExceedingToolValue := boPreventLimitSpeedExceeding.Value;

                  
END_GET
END_PROPERTY

METHOD InitializeCanSignals
                  i16Ibatt_ist.AppScalingDivisor :=1;
i16Ibatt_ist.AppScalingMultiplier :=1;
i16Ibatt_ist.AppScalingOffset :=0;
i16Ibatt_ist.AppUnit :="";
i16Ibatt_ist.CanDefault :=0;
i16Ibatt_ist.CanInit :=0;
i16Ibatt_ist.CanMax :=VBasic.LibConst.I16_MAX;
i16Ibatt_ist.CanMin :=VBasic.LibConst.I16_MIN;
i16Ibatt_ist.CanUnit :="";
i16Ibatt_ist.Description :="new signal";
i16Ibatt_ist.ErrorReaction := eErrorReaction.ERSIG_DFLT;
i16Ibatt_ist.ReceiverAdress :=1;
i16Ibatt_ist.ToolScalingDivisor :=1;
i16Ibatt_ist.ToolScalingMultiplier :=1;
i16Ibatt_ist.ToolScalingOffset :=0;
i16Ibatt_ist.ToolUnit :="";

u16Vbatt_ist.AppScalingDivisor :=1;
u16Vbatt_ist.AppScalingMultiplier :=1;
u16Vbatt_ist.AppScalingOffset :=0;
u16Vbatt_ist.AppUnit :="";
u16Vbatt_ist.CanDefault :=0;
u16Vbatt_ist.CanInit :=0;
u16Vbatt_ist.CanMax :=VBasic.LibConst.U16_MAX;
u16Vbatt_ist.CanMin :=VBasic.LibConst.U16_MIN;
u16Vbatt_ist.CanUnit :="";
u16Vbatt_ist.Description :="new signal";
u16Vbatt_ist.ErrorReaction := eErrorReaction.ERSIG_DFLT;
u16Vbatt_ist.ReceiverAdress :=1;
u16Vbatt_ist.ToolScalingDivisor :=1;
u16Vbatt_ist.ToolScalingMultiplier :=1;
u16Vbatt_ist.ToolScalingOffset :=0;
u16Vbatt_ist.ToolUnit :="";

u8Batt_Soc.AppScalingDivisor :=1;
u8Batt_Soc.AppScalingMultiplier :=1;
u8Batt_Soc.AppScalingOffset :=0;
u8Batt_Soc.AppUnit :="";
u8Batt_Soc.CanDefault :=0;
u8Batt_Soc.CanInit :=0;
u8Batt_Soc.CanMax :=VBasic.LibConst.U8_MAX;
u8Batt_Soc.CanMin :=VBasic.LibConst.U8_MIN;
u8Batt_Soc.CanUnit :="";
u8Batt_Soc.Description :="new signal";
u8Batt_Soc.ErrorReaction := eErrorReaction.ERSIG_DFLT;
u8Batt_Soc.ReceiverAdress :=1;
u8Batt_Soc.ToolScalingDivisor :=1;
u8Batt_Soc.ToolScalingMultiplier :=1;
u8Batt_Soc.ToolScalingOffset :=0;
u8Batt_Soc.ToolUnit :="";

boAddParkBrakeActive.AppScalingDivisor :=1;
boAddParkBrakeActive.AppScalingMultiplier :=1;
boAddParkBrakeActive.AppScalingOffset :=0;
boAddParkBrakeActive.AppUnit :="";
boAddParkBrakeActive.CanDefault :=0;
boAddParkBrakeActive.CanInit :=0;
boAddParkBrakeActive.CanMax :=1;
boAddParkBrakeActive.CanMin :=0;
boAddParkBrakeActive.CanUnit :="";
boAddParkBrakeActive.Description :="new signal";
boAddParkBrakeActive.ErrorReaction := eErrorReaction.ERSIG_DFLT;
boAddParkBrakeActive.ReceiverAdress :=1;
boAddParkBrakeActive.ToolScalingDivisor :=1;
boAddParkBrakeActive.ToolScalingMultiplier :=1;
boAddParkBrakeActive.ToolScalingOffset :=0;
boAddParkBrakeActive.ToolUnit :="";

boPreventLimitSpeedExceeding.AppScalingDivisor :=1;
boPreventLimitSpeedExceeding.AppScalingMultiplier :=1;
boPreventLimitSpeedExceeding.AppScalingOffset :=0;
boPreventLimitSpeedExceeding.AppUnit :="";
boPreventLimitSpeedExceeding.CanDefault :=0;
boPreventLimitSpeedExceeding.CanInit :=0;
boPreventLimitSpeedExceeding.CanMax :=1;
boPreventLimitSpeedExceeding.CanMin :=0;
boPreventLimitSpeedExceeding.CanUnit :="";
boPreventLimitSpeedExceeding.Description :="new signal";
boPreventLimitSpeedExceeding.ErrorReaction := eErrorReaction.ERSIG_DFLT;
boPreventLimitSpeedExceeding.ReceiverAdress :=1;
boPreventLimitSpeedExceeding.ToolScalingDivisor :=1;
boPreventLimitSpeedExceeding.ToolScalingMultiplier :=1;
boPreventLimitSpeedExceeding.ToolScalingOffset :=0;
boPreventLimitSpeedExceeding.ToolUnit :="";


                
END_METHOD
END_FUNCTION_BLOCK

FUNCTION_BLOCK Msg15C0SendToEvision7MessageClass EXTENDS CanReceiveMessageClass
  VAR_INPUT
    i16ElectricPumpPressureValue : Int16CanSignalClass;
    u16PvgTransRailElectricVoltage : UInt16CanSignalClass;
    boRelayCutOffVariatorElectricCmd : BoolCanSignalClass;
    boRelayEnableBatteryCmd : BoolCanSignalClass;
    boPictoAskResartController : BoolCanSignalClass;
    boPictoReloadBatteryImpossible : BoolCanSignalClass;
    u8Controller_FaultCode : UInt8CanSignalClass;
    u16Controller_FaultSubCode : UInt16CanSignalClass;
    Counter : UInt32CanSignalClass;
  END_VAR

            
          

METHOD SetData
  VAR_INPUT
    CanMsgPointer : POINTER TO CanMessageClass;
  END_VAR
                  IF IsValidPointer(canMsgPointer,'SetData') THEN
	SUPER^.SetData(CanMsgPointer);
	//Set the new data
	i16ElectricPumpPressureValue.Value := canMsgPointer^.GetInt16(0);
	u16PvgTransRailElectricVoltage.Value := canMsgPointer^.GetUint16(16);
	boRelayCutOffVariatorElectricCmd.Value := canMsgPointer^.GetBoolOnBit(32);
	boRelayEnableBatteryCmd.Value := canMsgPointer^.GetBoolOnBit(33);
	boPictoAskResartController.Value := canMsgPointer^.GetBoolOnBit(34);
	boPictoReloadBatteryImpossible.Value := canMsgPointer^.GetBoolOnBit(35);
	u8Controller_FaultCode.Value := canMsgPointer^.GetUint8(40);
	u16Controller_FaultSubCode.Value := canMsgPointer^.GetUint16(48);
	//And increase the counter
	Counter.Value := CanMsgPointer^.Counter.Value;
END_IF

                
END_METHOD

PROPERTY i16ElectricPumpPressureValueRawValue : INT
GET
                    IF i16ElectricPumpPressureValue.AppScalingMultiplier = 0 THEN
	_MatchLog^.Error("Get i16ElectricPumpPressureValueRawValue", "Division by Zero!");
	RETURN;
End_IF

i16ElectricPumpPressureValueRawValue := TO_INT((i16ElectricPumpPressureValue.Value - i16ElectricPumpPressureValue.AppScalingOffset) * i16ElectricPumpPressureValue.AppScalingDivisor / i16ElectricPumpPressureValue.AppScalingMultiplier);

                  
END_GET
END_PROPERTY

PROPERTY u16PvgTransRailElectricVoltageRawValue : UINT
GET
                    IF u16PvgTransRailElectricVoltage.AppScalingMultiplier = 0 THEN
	_MatchLog^.Error("Get u16PvgTransRailElectricVoltageRawValue", "Division by Zero!");
	RETURN;
End_IF

u16PvgTransRailElectricVoltageRawValue := TO_UINT((u16PvgTransRailElectricVoltage.Value - u16PvgTransRailElectricVoltage.AppScalingOffset) * u16PvgTransRailElectricVoltage.AppScalingDivisor / u16PvgTransRailElectricVoltage.AppScalingMultiplier);

                  
END_GET
END_PROPERTY

PROPERTY boRelayCutOffVariatorElectricCmdRawValue : BOOL
GET
                    boRelayCutOffVariatorElectricCmdRawValue := boRelayCutOffVariatorElectricCmd.Value;

                  
END_GET
END_PROPERTY

PROPERTY boRelayEnableBatteryCmdRawValue : BOOL
GET
                    boRelayEnableBatteryCmdRawValue := boRelayEnableBatteryCmd.Value;

                  
END_GET
END_PROPERTY

PROPERTY boPictoAskResartControllerRawValue : BOOL
GET
                    boPictoAskResartControllerRawValue := boPictoAskResartController.Value;

                  
END_GET
END_PROPERTY

PROPERTY boPictoReloadBatteryImpossibleRawValue : BOOL
GET
                    boPictoReloadBatteryImpossibleRawValue := boPictoReloadBatteryImpossible.Value;

                  
END_GET
END_PROPERTY

PROPERTY u8Controller_FaultCodeRawValue : USINT
GET
                    IF u8Controller_FaultCode.AppScalingMultiplier = 0 THEN
	_MatchLog^.Error("Get u8Controller_FaultCodeRawValue", "Division by Zero!");
	RETURN;
End_IF

u8Controller_FaultCodeRawValue := TO_USINT((u8Controller_FaultCode.Value - u8Controller_FaultCode.AppScalingOffset) * u8Controller_FaultCode.AppScalingDivisor / u8Controller_FaultCode.AppScalingMultiplier);

                  
END_GET
END_PROPERTY

PROPERTY u16Controller_FaultSubCodeRawValue : UINT
GET
                    IF u16Controller_FaultSubCode.AppScalingMultiplier = 0 THEN
	_MatchLog^.Error("Get u16Controller_FaultSubCodeRawValue", "Division by Zero!");
	RETURN;
End_IF

u16Controller_FaultSubCodeRawValue := TO_UINT((u16Controller_FaultSubCode.Value - u16Controller_FaultSubCode.AppScalingOffset) * u16Controller_FaultSubCode.AppScalingDivisor / u16Controller_FaultSubCode.AppScalingMultiplier);

                  
END_GET
END_PROPERTY

PROPERTY i16ElectricPumpPressureValueToolValue : INT
GET
                    IF i16ElectricPumpPressureValue.ToolScalingDivisor = 0 OR i16ElectricPumpPressureValue.AppScalingMultiplier = 0 THEN
	_MatchLog^.Error("Get i16ElectricPumpPressureValueToolValue", "Division by Zero!");
	RETURN;
END_IF

i16ElectricPumpPressureValueToolValue := TO_INT(((i16ElectricPumpPressureValue.Value - i16ElectricPumpPressureValue.AppScalingOffset) * i16ElectricPumpPressureValue.AppScalingDivisor / i16ElectricPumpPressureValue.AppScalingMultiplier * i16ElectricPumpPressureValue.ToolScalingMultiplier / i16ElectricPumpPressureValue.ToolScalingDivisor) + i16ElectricPumpPressureValue.ToolScalingOffset);

                  
END_GET
END_PROPERTY

PROPERTY u16PvgTransRailElectricVoltageToolValue : UINT
GET
                    IF u16PvgTransRailElectricVoltage.ToolScalingDivisor = 0 OR u16PvgTransRailElectricVoltage.AppScalingMultiplier = 0 THEN
	_MatchLog^.Error("Get u16PvgTransRailElectricVoltageToolValue", "Division by Zero!");
	RETURN;
END_IF

u16PvgTransRailElectricVoltageToolValue := TO_UINT(((u16PvgTransRailElectricVoltage.Value - u16PvgTransRailElectricVoltage.AppScalingOffset) * u16PvgTransRailElectricVoltage.AppScalingDivisor / u16PvgTransRailElectricVoltage.AppScalingMultiplier * u16PvgTransRailElectricVoltage.ToolScalingMultiplier / u16PvgTransRailElectricVoltage.ToolScalingDivisor) + u16PvgTransRailElectricVoltage.ToolScalingOffset);

                  
END_GET
END_PROPERTY

PROPERTY boRelayCutOffVariatorElectricCmdToolValue : BOOL
GET
                    boRelayCutOffVariatorElectricCmdToolValue := boRelayCutOffVariatorElectricCmd.Value;

                  
END_GET
END_PROPERTY

PROPERTY boRelayEnableBatteryCmdToolValue : BOOL
GET
                    boRelayEnableBatteryCmdToolValue := boRelayEnableBatteryCmd.Value;

                  
END_GET
END_PROPERTY

PROPERTY boPictoAskResartControllerToolValue : BOOL
GET
                    boPictoAskResartControllerToolValue := boPictoAskResartController.Value;

                  
END_GET
END_PROPERTY

PROPERTY boPictoReloadBatteryImpossibleToolValue : BOOL
GET
                    boPictoReloadBatteryImpossibleToolValue := boPictoReloadBatteryImpossible.Value;

                  
END_GET
END_PROPERTY

PROPERTY u8Controller_FaultCodeToolValue : USINT
GET
                    IF u8Controller_FaultCode.ToolScalingDivisor = 0 OR u8Controller_FaultCode.AppScalingMultiplier = 0 THEN
	_MatchLog^.Error("Get u8Controller_FaultCodeToolValue", "Division by Zero!");
	RETURN;
END_IF

u8Controller_FaultCodeToolValue := TO_USINT(((u8Controller_FaultCode.Value - u8Controller_FaultCode.AppScalingOffset) * u8Controller_FaultCode.AppScalingDivisor / u8Controller_FaultCode.AppScalingMultiplier * u8Controller_FaultCode.ToolScalingMultiplier / u8Controller_FaultCode.ToolScalingDivisor) + u8Controller_FaultCode.ToolScalingOffset);

                  
END_GET
END_PROPERTY

PROPERTY u16Controller_FaultSubCodeToolValue : UINT
GET
                    IF u16Controller_FaultSubCode.ToolScalingDivisor = 0 OR u16Controller_FaultSubCode.AppScalingMultiplier = 0 THEN
	_MatchLog^.Error("Get u16Controller_FaultSubCodeToolValue", "Division by Zero!");
	RETURN;
END_IF

u16Controller_FaultSubCodeToolValue := TO_UINT(((u16Controller_FaultSubCode.Value - u16Controller_FaultSubCode.AppScalingOffset) * u16Controller_FaultSubCode.AppScalingDivisor / u16Controller_FaultSubCode.AppScalingMultiplier * u16Controller_FaultSubCode.ToolScalingMultiplier / u16Controller_FaultSubCode.ToolScalingDivisor) + u16Controller_FaultSubCode.ToolScalingOffset);

                  
END_GET
END_PROPERTY

METHOD InitializeCanSignals
                  i16ElectricPumpPressureValue.AppScalingDivisor :=1;
i16ElectricPumpPressureValue.AppScalingMultiplier :=1;
i16ElectricPumpPressureValue.AppScalingOffset :=0;
i16ElectricPumpPressureValue.AppUnit :="";
i16ElectricPumpPressureValue.CanDefault :=0;
i16ElectricPumpPressureValue.CanInit :=0;
i16ElectricPumpPressureValue.CanMax :=VBasic.LibConst.I16_MAX;
i16ElectricPumpPressureValue.CanMin :=VBasic.LibConst.I16_MIN;
i16ElectricPumpPressureValue.CanUnit :="";
i16ElectricPumpPressureValue.Description :="new signal";
i16ElectricPumpPressureValue.ErrorReaction := eErrorReaction.ERSIG_DFLT;
i16ElectricPumpPressureValue.ReceiverAdress :=1;
i16ElectricPumpPressureValue.ToolScalingDivisor :=1;
i16ElectricPumpPressureValue.ToolScalingMultiplier :=1;
i16ElectricPumpPressureValue.ToolScalingOffset :=0;
i16ElectricPumpPressureValue.ToolUnit :="";

u16PvgTransRailElectricVoltage.AppScalingDivisor :=1;
u16PvgTransRailElectricVoltage.AppScalingMultiplier :=1;
u16PvgTransRailElectricVoltage.AppScalingOffset :=0;
u16PvgTransRailElectricVoltage.AppUnit :="";
u16PvgTransRailElectricVoltage.CanDefault :=0;
u16PvgTransRailElectricVoltage.CanInit :=0;
u16PvgTransRailElectricVoltage.CanMax :=VBasic.LibConst.U16_MAX;
u16PvgTransRailElectricVoltage.CanMin :=VBasic.LibConst.U16_MIN;
u16PvgTransRailElectricVoltage.CanUnit :="";
u16PvgTransRailElectricVoltage.Description :="new signal";
u16PvgTransRailElectricVoltage.ErrorReaction := eErrorReaction.ERSIG_DFLT;
u16PvgTransRailElectricVoltage.ReceiverAdress :=1;
u16PvgTransRailElectricVoltage.ToolScalingDivisor :=1;
u16PvgTransRailElectricVoltage.ToolScalingMultiplier :=1;
u16PvgTransRailElectricVoltage.ToolScalingOffset :=0;
u16PvgTransRailElectricVoltage.ToolUnit :="";

boRelayCutOffVariatorElectricCmd.AppScalingDivisor :=1;
boRelayCutOffVariatorElectricCmd.AppScalingMultiplier :=1;
boRelayCutOffVariatorElectricCmd.AppScalingOffset :=0;
boRelayCutOffVariatorElectricCmd.AppUnit :="";
boRelayCutOffVariatorElectricCmd.CanDefault :=0;
boRelayCutOffVariatorElectricCmd.CanInit :=0;
boRelayCutOffVariatorElectricCmd.CanMax :=1;
boRelayCutOffVariatorElectricCmd.CanMin :=0;
boRelayCutOffVariatorElectricCmd.CanUnit :="";
boRelayCutOffVariatorElectricCmd.Description :="new signal";
boRelayCutOffVariatorElectricCmd.ErrorReaction := eErrorReaction.ERSIG_DFLT;
boRelayCutOffVariatorElectricCmd.ReceiverAdress :=1;
boRelayCutOffVariatorElectricCmd.ToolScalingDivisor :=1;
boRelayCutOffVariatorElectricCmd.ToolScalingMultiplier :=1;
boRelayCutOffVariatorElectricCmd.ToolScalingOffset :=0;
boRelayCutOffVariatorElectricCmd.ToolUnit :="";

boRelayEnableBatteryCmd.AppScalingDivisor :=1;
boRelayEnableBatteryCmd.AppScalingMultiplier :=1;
boRelayEnableBatteryCmd.AppScalingOffset :=0;
boRelayEnableBatteryCmd.AppUnit :="";
boRelayEnableBatteryCmd.CanDefault :=0;
boRelayEnableBatteryCmd.CanInit :=0;
boRelayEnableBatteryCmd.CanMax :=1;
boRelayEnableBatteryCmd.CanMin :=0;
boRelayEnableBatteryCmd.CanUnit :="";
boRelayEnableBatteryCmd.Description :="new signal";
boRelayEnableBatteryCmd.ErrorReaction := eErrorReaction.ERSIG_DFLT;
boRelayEnableBatteryCmd.ReceiverAdress :=1;
boRelayEnableBatteryCmd.ToolScalingDivisor :=1;
boRelayEnableBatteryCmd.ToolScalingMultiplier :=1;
boRelayEnableBatteryCmd.ToolScalingOffset :=0;
boRelayEnableBatteryCmd.ToolUnit :="";

boPictoAskResartController.AppScalingDivisor :=1;
boPictoAskResartController.AppScalingMultiplier :=1;
boPictoAskResartController.AppScalingOffset :=0;
boPictoAskResartController.AppUnit :="";
boPictoAskResartController.CanDefault :=0;
boPictoAskResartController.CanInit :=0;
boPictoAskResartController.CanMax :=1;
boPictoAskResartController.CanMin :=0;
boPictoAskResartController.CanUnit :="";
boPictoAskResartController.Description :="new signal";
boPictoAskResartController.ErrorReaction := eErrorReaction.ERSIG_DFLT;
boPictoAskResartController.ReceiverAdress :=1;
boPictoAskResartController.ToolScalingDivisor :=1;
boPictoAskResartController.ToolScalingMultiplier :=1;
boPictoAskResartController.ToolScalingOffset :=0;
boPictoAskResartController.ToolUnit :="";

boPictoReloadBatteryImpossible.AppScalingDivisor :=1;
boPictoReloadBatteryImpossible.AppScalingMultiplier :=1;
boPictoReloadBatteryImpossible.AppScalingOffset :=0;
boPictoReloadBatteryImpossible.AppUnit :="";
boPictoReloadBatteryImpossible.CanDefault :=0;
boPictoReloadBatteryImpossible.CanInit :=0;
boPictoReloadBatteryImpossible.CanMax :=1;
boPictoReloadBatteryImpossible.CanMin :=0;
boPictoReloadBatteryImpossible.CanUnit :="";
boPictoReloadBatteryImpossible.Description :="new signal";
boPictoReloadBatteryImpossible.ErrorReaction := eErrorReaction.ERSIG_DFLT;
boPictoReloadBatteryImpossible.ReceiverAdress :=1;
boPictoReloadBatteryImpossible.ToolScalingDivisor :=1;
boPictoReloadBatteryImpossible.ToolScalingMultiplier :=1;
boPictoReloadBatteryImpossible.ToolScalingOffset :=0;
boPictoReloadBatteryImpossible.ToolUnit :="";

u8Controller_FaultCode.AppScalingDivisor :=1;
u8Controller_FaultCode.AppScalingMultiplier :=1;
u8Controller_FaultCode.AppScalingOffset :=0;
u8Controller_FaultCode.AppUnit :="";
u8Controller_FaultCode.CanDefault :=0;
u8Controller_FaultCode.CanInit :=0;
u8Controller_FaultCode.CanMax :=VBasic.LibConst.U8_MAX;
u8Controller_FaultCode.CanMin :=VBasic.LibConst.U8_MIN;
u8Controller_FaultCode.CanUnit :="";
u8Controller_FaultCode.Description :="new signal";
u8Controller_FaultCode.ErrorReaction := eErrorReaction.ERSIG_DFLT;
u8Controller_FaultCode.ReceiverAdress :=1;
u8Controller_FaultCode.ToolScalingDivisor :=1;
u8Controller_FaultCode.ToolScalingMultiplier :=1;
u8Controller_FaultCode.ToolScalingOffset :=0;
u8Controller_FaultCode.ToolUnit :="";

u16Controller_FaultSubCode.AppScalingDivisor :=1;
u16Controller_FaultSubCode.AppScalingMultiplier :=1;
u16Controller_FaultSubCode.AppScalingOffset :=0;
u16Controller_FaultSubCode.AppUnit :="";
u16Controller_FaultSubCode.CanDefault :=0;
u16Controller_FaultSubCode.CanInit :=0;
u16Controller_FaultSubCode.CanMax :=VBasic.LibConst.U16_MAX;
u16Controller_FaultSubCode.CanMin :=VBasic.LibConst.U16_MIN;
u16Controller_FaultSubCode.CanUnit :="";
u16Controller_FaultSubCode.Description :="new signal";
u16Controller_FaultSubCode.ErrorReaction := eErrorReaction.ERSIG_DFLT;
u16Controller_FaultSubCode.ReceiverAdress :=1;
u16Controller_FaultSubCode.ToolScalingDivisor :=1;
u16Controller_FaultSubCode.ToolScalingMultiplier :=1;
u16Controller_FaultSubCode.ToolScalingOffset :=0;
u16Controller_FaultSubCode.ToolUnit :="";


                
END_METHOD
END_FUNCTION_BLOCK

FUNCTION_BLOCK MsgDebugC0SendToEvision7MessageClass EXTENDS CanReceiveMessageClass
  VAR_INPUT
    u16FaultyValue : UInt16CanSignalClass;
    u8DeviceNum : UInt8CanSignalClass;
    u8ErrorCode : UInt8CanSignalClass;
    Counter : UInt32CanSignalClass;
  END_VAR

            
          

METHOD SetData
  VAR_INPUT
    CanMsgPointer : POINTER TO CanMessageClass;
  END_VAR
                  IF IsValidPointer(canMsgPointer,'SetData') THEN
	SUPER^.SetData(CanMsgPointer);
	//Set the new data
	u16FaultyValue.Value := canMsgPointer^.GetUint16(0);
	u8DeviceNum.Value := canMsgPointer^.GetUint8(16);
	u8ErrorCode.Value := canMsgPointer^.GetUint8(24);
	//And increase the counter
	Counter.Value := CanMsgPointer^.Counter.Value;
END_IF

                
END_METHOD

PROPERTY u16FaultyValueRawValue : UINT
GET
                    IF u16FaultyValue.AppScalingMultiplier = 0 THEN
	_MatchLog^.Error("Get u16FaultyValueRawValue", "Division by Zero!");
	RETURN;
End_IF

u16FaultyValueRawValue := TO_UINT((u16FaultyValue.Value - u16FaultyValue.AppScalingOffset) * u16FaultyValue.AppScalingDivisor / u16FaultyValue.AppScalingMultiplier);

                  
END_GET
END_PROPERTY

PROPERTY u8DeviceNumRawValue : USINT
GET
                    IF u8DeviceNum.AppScalingMultiplier = 0 THEN
	_MatchLog^.Error("Get u8DeviceNumRawValue", "Division by Zero!");
	RETURN;
End_IF

u8DeviceNumRawValue := TO_USINT((u8DeviceNum.Value - u8DeviceNum.AppScalingOffset) * u8DeviceNum.AppScalingDivisor / u8DeviceNum.AppScalingMultiplier);

                  
END_GET
END_PROPERTY

PROPERTY u8ErrorCodeRawValue : USINT
GET
                    IF u8ErrorCode.AppScalingMultiplier = 0 THEN
	_MatchLog^.Error("Get u8ErrorCodeRawValue", "Division by Zero!");
	RETURN;
End_IF

u8ErrorCodeRawValue := TO_USINT((u8ErrorCode.Value - u8ErrorCode.AppScalingOffset) * u8ErrorCode.AppScalingDivisor / u8ErrorCode.AppScalingMultiplier);

                  
END_GET
END_PROPERTY

PROPERTY u16FaultyValueToolValue : UINT
GET
                    IF u16FaultyValue.ToolScalingDivisor = 0 OR u16FaultyValue.AppScalingMultiplier = 0 THEN
	_MatchLog^.Error("Get u16FaultyValueToolValue", "Division by Zero!");
	RETURN;
END_IF

u16FaultyValueToolValue := TO_UINT(((u16FaultyValue.Value - u16FaultyValue.AppScalingOffset) * u16FaultyValue.AppScalingDivisor / u16FaultyValue.AppScalingMultiplier * u16FaultyValue.ToolScalingMultiplier / u16FaultyValue.ToolScalingDivisor) + u16FaultyValue.ToolScalingOffset);

                  
END_GET
END_PROPERTY

PROPERTY u8DeviceNumToolValue : USINT
GET
                    IF u8DeviceNum.ToolScalingDivisor = 0 OR u8DeviceNum.AppScalingMultiplier = 0 THEN
	_MatchLog^.Error("Get u8DeviceNumToolValue", "Division by Zero!");
	RETURN;
END_IF

u8DeviceNumToolValue := TO_USINT(((u8DeviceNum.Value - u8DeviceNum.AppScalingOffset) * u8DeviceNum.AppScalingDivisor / u8DeviceNum.AppScalingMultiplier * u8DeviceNum.ToolScalingMultiplier / u8DeviceNum.ToolScalingDivisor) + u8DeviceNum.ToolScalingOffset);

                  
END_GET
END_PROPERTY

PROPERTY u8ErrorCodeToolValue : USINT
GET
                    IF u8ErrorCode.ToolScalingDivisor = 0 OR u8ErrorCode.AppScalingMultiplier = 0 THEN
	_MatchLog^.Error("Get u8ErrorCodeToolValue", "Division by Zero!");
	RETURN;
END_IF

u8ErrorCodeToolValue := TO_USINT(((u8ErrorCode.Value - u8ErrorCode.AppScalingOffset) * u8ErrorCode.AppScalingDivisor / u8ErrorCode.AppScalingMultiplier * u8ErrorCode.ToolScalingMultiplier / u8ErrorCode.ToolScalingDivisor) + u8ErrorCode.ToolScalingOffset);

                  
END_GET
END_PROPERTY

METHOD InitializeCanSignals
                  u16FaultyValue.AppScalingDivisor :=1;
u16FaultyValue.AppScalingMultiplier :=1;
u16FaultyValue.AppScalingOffset :=0;
u16FaultyValue.AppUnit :="";
u16FaultyValue.CanDefault :=0;
u16FaultyValue.CanInit :=0;
u16FaultyValue.CanMax :=VBasic.LibConst.U16_MAX;
u16FaultyValue.CanMin :=VBasic.LibConst.U16_MIN;
u16FaultyValue.CanUnit :="";
u16FaultyValue.Description :="";
u16FaultyValue.ErrorReaction := eErrorReaction.ERSIG_DFLT;
u16FaultyValue.ReceiverAdress :=1;
u16FaultyValue.ToolScalingDivisor :=1;
u16FaultyValue.ToolScalingMultiplier :=1;
u16FaultyValue.ToolScalingOffset :=0;
u16FaultyValue.ToolUnit :="";

u8DeviceNum.AppScalingDivisor :=1;
u8DeviceNum.AppScalingMultiplier :=1;
u8DeviceNum.AppScalingOffset :=0;
u8DeviceNum.AppUnit :="";
u8DeviceNum.CanDefault :=0;
u8DeviceNum.CanInit :=0;
u8DeviceNum.CanMax :=VBasic.LibConst.U8_MAX;
u8DeviceNum.CanMin :=VBasic.LibConst.U8_MIN;
u8DeviceNum.CanUnit :="";
u8DeviceNum.Description :="";
u8DeviceNum.ErrorReaction := eErrorReaction.ERSIG_DFLT;
u8DeviceNum.ReceiverAdress :=1;
u8DeviceNum.ToolScalingDivisor :=1;
u8DeviceNum.ToolScalingMultiplier :=1;
u8DeviceNum.ToolScalingOffset :=0;
u8DeviceNum.ToolUnit :="";

u8ErrorCode.AppScalingDivisor :=1;
u8ErrorCode.AppScalingMultiplier :=1;
u8ErrorCode.AppScalingOffset :=0;
u8ErrorCode.AppUnit :="";
u8ErrorCode.CanDefault :=0;
u8ErrorCode.CanInit :=0;
u8ErrorCode.CanMax :=VBasic.LibConst.U8_MAX;
u8ErrorCode.CanMin :=VBasic.LibConst.U8_MIN;
u8ErrorCode.CanUnit :="";
u8ErrorCode.Description :="";
u8ErrorCode.ErrorReaction := eErrorReaction.ERSIG_DFLT;
u8ErrorCode.ReceiverAdress :=1;
u8ErrorCode.ToolScalingDivisor :=1;
u8ErrorCode.ToolScalingMultiplier :=1;
u8ErrorCode.ToolScalingOffset :=0;
u8ErrorCode.ToolUnit :="";


                
END_METHOD
END_FUNCTION_BLOCK

FUNCTION_BLOCK Msg1C1SendToEvision7MessageClass EXTENDS CanReceiveMessageClass
  VAR_INPUT
    bogBattery_On_Off : BoolCanSignalClass;
    bogPreheat_On_Off : BoolCanSignalClass;
    bogEngine_Faillure_On_Off : BoolCanSignalClass;
    bogMaintenance_On_Off : BoolCanSignalClass;
    bogOil_On_OFF : BoolCanSignalClass;
    bogDeltaArmSectorDown : BoolCanSignalClass;
    bogArrowArmSectorDown : BoolCanSignalClass;
    bogPendularSectorDown : BoolCanSignalClass;
    bogDeltaArmInCenter : BoolCanSignalClass;
    bogArrowArmInCenter : BoolCanSignalClass;
    bogPendularInCenter : BoolCanSignalClass;
    bogBasketRotationInCenter : BoolCanSignalClass;
    bogTelescopeInCenter : BoolCanSignalClass;
    bogBasketInclinaisonInCenter : BoolCanSignalClass;
    bogDeltaArmMoveUpAllow : BoolCanSignalClass;
    bogDeltaArmMoveDownAllow : BoolCanSignalClass;
    bogArrowArmMoveUpAllow : BoolCanSignalClass;
    bogArrowArmMoveDownAllow : BoolCanSignalClass;
    bogPendularMoveUpAllow : BoolCanSignalClass;
    bogPendularMoveDownAllow : BoolCanSignalClass;
    bogTelescopeMoveOutAllow : BoolCanSignalClass;
    bogTelescopeMoveInAllow : BoolCanSignalClass;
    bogTurretCtClockWiseMoveAllow : BoolCanSignalClass;
    bogTurretClockWiseMoveAllow : BoolCanSignalClass;
    bogBasketRotCtClockWiseMoveAllow : BoolCanSignalClass;
    bogBasketRotClockWiseMoveAllow : BoolCanSignalClass;
    bogBasketInclinMoveUpAllow : BoolCanSignalClass;
    bogBasketInclinMoveDownAllow : BoolCanSignalClass;
    bogVehiculeDefault : BoolCanSignalClass;
    bogTelescopeOutputPossible : BoolCanSignalClass;
    bogTelescopeWinderFault : BoolCanSignalClass;
    bogNacellePostSelector : BoolCanSignalClass;
    bogSTOP_On_Off : BoolCanSignalClass;
    bogSafeManSystem : BoolCanSignalClass;
    bogHighSpeedAllow : BoolCanSignalClass;
    bogAutomatiqueStop : BoolCanSignalClass;
    bogLowSpeedByFault : BoolCanSignalClass;
    bogMeasuringMastFault : BoolCanSignalClass;
    bogMeasuringMatOption : BoolCanSignalClass;
    bogBasketAccessLocked : BoolCanSignalClass;
    bogFilterOverloadNoActive : BoolCanSignalClass;
    bogAnticlockwiseBasketSlew : BoolCanSignalClass;
    bogClockwiseBasketSlew : BoolCanSignalClass;
    bogFlashLightForced : BoolCanSignalClass;
    bogBasketAccessLockOption : BoolCanSignalClass;
    bogBasketLateralStopOption : BoolCanSignalClass;
    bogBasketStepClosed : BoolCanSignalClass;
    bogSystemFault : BoolCanSignalClass;
    bogTrans1PressureSensorFault : BoolCanSignalClass;
    bogTrans2PressureSensorFault : BoolCanSignalClass;
    bogOverloadSecurity : BoolCanSignalClass;
    bogDeltaArmJoysCenteredTeles : BoolCanSignalClass;
    bogArrowJoystickCenteredTurret : BoolCanSignalClass;
    bogDeltaArmMoveUp : BoolCanSignalClass;
    bogDeltaArmMoveDown : BoolCanSignalClass;
    bogArrowArmMoveUp : BoolCanSignalClass;
    bogArrowArmMoveDown : BoolCanSignalClass;
    bogTelescopeMoveOut : BoolCanSignalClass;
    bogTelescopeMoveIn : BoolCanSignalClass;
    bogTurretCounterClockWiseMove : BoolCanSignalClass;
    bogTurretClockWiseMove : BoolCanSignalClass;
    bogTurretEncoderFault : BoolCanSignalClass;
    bogGeneratorOption : BoolCanSignalClass;
    bogGeneratorActive : BoolCanSignalClass;
    Counter : UInt32CanSignalClass;
  END_VAR

            
          

METHOD SetData
  VAR_INPUT
    CanMsgPointer : POINTER TO CanMessageClass;
  END_VAR
                  IF IsValidPointer(canMsgPointer,'SetData') THEN
	SUPER^.SetData(CanMsgPointer);
	//Set the new data
	bogBattery_On_Off.Value := canMsgPointer^.GetBoolOnBit(0);
	bogPreheat_On_Off.Value := canMsgPointer^.GetBoolOnBit(1);
	bogEngine_Faillure_On_Off.Value := canMsgPointer^.GetBoolOnBit(2);
	bogMaintenance_On_Off.Value := canMsgPointer^.GetBoolOnBit(3);
	bogOil_On_OFF.Value := canMsgPointer^.GetBoolOnBit(4);
	bogDeltaArmSectorDown.Value := canMsgPointer^.GetBoolOnBit(5);
	bogArrowArmSectorDown.Value := canMsgPointer^.GetBoolOnBit(6);
	bogPendularSectorDown.Value := canMsgPointer^.GetBoolOnBit(7);
	bogDeltaArmInCenter.Value := canMsgPointer^.GetBoolOnBit(8);
	bogArrowArmInCenter.Value := canMsgPointer^.GetBoolOnBit(9);
	bogPendularInCenter.Value := canMsgPointer^.GetBoolOnBit(10);
	bogBasketRotationInCenter.Value := canMsgPointer^.GetBoolOnBit(11);
	bogTelescopeInCenter.Value := canMsgPointer^.GetBoolOnBit(12);
	bogBasketInclinaisonInCenter.Value := canMsgPointer^.GetBoolOnBit(13);
	bogDeltaArmMoveUpAllow.Value := canMsgPointer^.GetBoolOnBit(14);
	bogDeltaArmMoveDownAllow.Value := canMsgPointer^.GetBoolOnBit(15);
	bogArrowArmMoveUpAllow.Value := canMsgPointer^.GetBoolOnBit(16);
	bogArrowArmMoveDownAllow.Value := canMsgPointer^.GetBoolOnBit(17);
	bogPendularMoveUpAllow.Value := canMsgPointer^.GetBoolOnBit(18);
	bogPendularMoveDownAllow.Value := canMsgPointer^.GetBoolOnBit(19);
	bogTelescopeMoveOutAllow.Value := canMsgPointer^.GetBoolOnBit(20);
	bogTelescopeMoveInAllow.Value := canMsgPointer^.GetBoolOnBit(21);
	bogTurretCtClockWiseMoveAllow.Value := canMsgPointer^.GetBoolOnBit(22);
	bogTurretClockWiseMoveAllow.Value := canMsgPointer^.GetBoolOnBit(23);
	bogBasketRotCtClockWiseMoveAllow.Value := canMsgPointer^.GetBoolOnBit(24);
	bogBasketRotClockWiseMoveAllow.Value := canMsgPointer^.GetBoolOnBit(25);
	bogBasketInclinMoveUpAllow.Value := canMsgPointer^.GetBoolOnBit(26);
	bogBasketInclinMoveDownAllow.Value := canMsgPointer^.GetBoolOnBit(27);
	bogVehiculeDefault.Value := canMsgPointer^.GetBoolOnBit(28);
	bogTelescopeOutputPossible.Value := canMsgPointer^.GetBoolOnBit(29);
	bogTelescopeWinderFault.Value := canMsgPointer^.GetBoolOnBit(30);
	bogNacellePostSelector.Value := canMsgPointer^.GetBoolOnBit(31);
	bogSTOP_On_Off.Value := canMsgPointer^.GetBoolOnBit(32);
	bogSafeManSystem.Value := canMsgPointer^.GetBoolOnBit(33);
	bogHighSpeedAllow.Value := canMsgPointer^.GetBoolOnBit(34);
	bogAutomatiqueStop.Value := canMsgPointer^.GetBoolOnBit(35);
	bogLowSpeedByFault.Value := canMsgPointer^.GetBoolOnBit(36);
	bogMeasuringMastFault.Value := canMsgPointer^.GetBoolOnBit(37);
	bogMeasuringMatOption.Value := canMsgPointer^.GetBoolOnBit(38);
	bogBasketAccessLocked.Value := canMsgPointer^.GetBoolOnBit(39);
	bogFilterOverloadNoActive.Value := canMsgPointer^.GetBoolOnBit(40);
	bogAnticlockwiseBasketSlew.Value := canMsgPointer^.GetBoolOnBit(41);
	bogClockwiseBasketSlew.Value := canMsgPointer^.GetBoolOnBit(42);
	bogFlashLightForced.Value := canMsgPointer^.GetBoolOnBit(43);
	bogBasketAccessLockOption.Value := canMsgPointer^.GetBoolOnBit(44);
	bogBasketLateralStopOption.Value := canMsgPointer^.GetBoolOnBit(45);
	bogBasketStepClosed.Value := canMsgPointer^.GetBoolOnBit(46);
	bogSystemFault.Value := canMsgPointer^.GetBoolOnBit(47);
	bogTrans1PressureSensorFault.Value := canMsgPointer^.GetBoolOnBit(48);
	bogTrans2PressureSensorFault.Value := canMsgPointer^.GetBoolOnBit(49);
	bogOverloadSecurity.Value := canMsgPointer^.GetBoolOnBit(50);
	bogDeltaArmJoysCenteredTeles.Value := canMsgPointer^.GetBoolOnBit(51);
	bogArrowJoystickCenteredTurret.Value := canMsgPointer^.GetBoolOnBit(52);
	bogDeltaArmMoveUp.Value := canMsgPointer^.GetBoolOnBit(53);
	bogDeltaArmMoveDown.Value := canMsgPointer^.GetBoolOnBit(54);
	bogArrowArmMoveUp.Value := canMsgPointer^.GetBoolOnBit(55);
	bogArrowArmMoveDown.Value := canMsgPointer^.GetBoolOnBit(56);
	bogTelescopeMoveOut.Value := canMsgPointer^.GetBoolOnBit(57);
	bogTelescopeMoveIn.Value := canMsgPointer^.GetBoolOnBit(58);
	bogTurretCounterClockWiseMove.Value := canMsgPointer^.GetBoolOnBit(59);
	bogTurretClockWiseMove.Value := canMsgPointer^.GetBoolOnBit(60);
	bogTurretEncoderFault.Value := canMsgPointer^.GetBoolOnBit(61);
	bogGeneratorOption.Value := canMsgPointer^.GetBoolOnBit(62);
	bogGeneratorActive.Value := canMsgPointer^.GetBoolOnBit(63);
	//And increase the counter
	Counter.Value := CanMsgPointer^.Counter.Value;
END_IF

                
END_METHOD

PROPERTY bogBattery_On_OffRawValue : BOOL
GET
                    bogBattery_On_OffRawValue := bogBattery_On_Off.Value;

                  
END_GET
END_PROPERTY

PROPERTY bogPreheat_On_OffRawValue : BOOL
GET
                    bogPreheat_On_OffRawValue := bogPreheat_On_Off.Value;

                  
END_GET
END_PROPERTY

PROPERTY bogEngine_Faillure_On_OffRawValue : BOOL
GET
                    bogEngine_Faillure_On_OffRawValue := bogEngine_Faillure_On_Off.Value;

                  
END_GET
END_PROPERTY

PROPERTY bogMaintenance_On_OffRawValue : BOOL
GET
                    bogMaintenance_On_OffRawValue := bogMaintenance_On_Off.Value;

                  
END_GET
END_PROPERTY

PROPERTY bogOil_On_OFFRawValue : BOOL
GET
                    bogOil_On_OFFRawValue := bogOil_On_OFF.Value;

                  
END_GET
END_PROPERTY

PROPERTY bogDeltaArmSectorDownRawValue : BOOL
GET
                    bogDeltaArmSectorDownRawValue := bogDeltaArmSectorDown.Value;

                  
END_GET
END_PROPERTY

PROPERTY bogArrowArmSectorDownRawValue : BOOL
GET
                    bogArrowArmSectorDownRawValue := bogArrowArmSectorDown.Value;

                  
END_GET
END_PROPERTY

PROPERTY bogPendularSectorDownRawValue : BOOL
GET
                    bogPendularSectorDownRawValue := bogPendularSectorDown.Value;

                  
END_GET
END_PROPERTY

PROPERTY bogDeltaArmInCenterRawValue : BOOL
GET
                    bogDeltaArmInCenterRawValue := bogDeltaArmInCenter.Value;

                  
END_GET
END_PROPERTY

PROPERTY bogArrowArmInCenterRawValue : BOOL
GET
                    bogArrowArmInCenterRawValue := bogArrowArmInCenter.Value;

                  
END_GET
END_PROPERTY

PROPERTY bogPendularInCenterRawValue : BOOL
GET
                    bogPendularInCenterRawValue := bogPendularInCenter.Value;

                  
END_GET
END_PROPERTY

PROPERTY bogBasketRotationInCenterRawValue : BOOL
GET
                    bogBasketRotationInCenterRawValue := bogBasketRotationInCenter.Value;

                  
END_GET
END_PROPERTY

PROPERTY bogTelescopeInCenterRawValue : BOOL
GET
                    bogTelescopeInCenterRawValue := bogTelescopeInCenter.Value;

                  
END_GET
END_PROPERTY

PROPERTY bogBasketInclinaisonInCenterRawValue : BOOL
GET
                    bogBasketInclinaisonInCenterRawValue := bogBasketInclinaisonInCenter.Value;

                  
END_GET
END_PROPERTY

PROPERTY bogDeltaArmMoveUpAllowRawValue : BOOL
GET
                    bogDeltaArmMoveUpAllowRawValue := bogDeltaArmMoveUpAllow.Value;

                  
END_GET
END_PROPERTY

PROPERTY bogDeltaArmMoveDownAllowRawValue : BOOL
GET
                    bogDeltaArmMoveDownAllowRawValue := bogDeltaArmMoveDownAllow.Value;

                  
END_GET
END_PROPERTY

PROPERTY bogArrowArmMoveUpAllowRawValue : BOOL
GET
                    bogArrowArmMoveUpAllowRawValue := bogArrowArmMoveUpAllow.Value;

                  
END_GET
END_PROPERTY

PROPERTY bogArrowArmMoveDownAllowRawValue : BOOL
GET
                    bogArrowArmMoveDownAllowRawValue := bogArrowArmMoveDownAllow.Value;

                  
END_GET
END_PROPERTY

PROPERTY bogPendularMoveUpAllowRawValue : BOOL
GET
                    bogPendularMoveUpAllowRawValue := bogPendularMoveUpAllow.Value;

                  
END_GET
END_PROPERTY

PROPERTY bogPendularMoveDownAllowRawValue : BOOL
GET
                    bogPendularMoveDownAllowRawValue := bogPendularMoveDownAllow.Value;

                  
END_GET
END_PROPERTY

PROPERTY bogTelescopeMoveOutAllowRawValue : BOOL
GET
                    bogTelescopeMoveOutAllowRawValue := bogTelescopeMoveOutAllow.Value;

                  
END_GET
END_PROPERTY

PROPERTY bogTelescopeMoveInAllowRawValue : BOOL
GET
                    bogTelescopeMoveInAllowRawValue := bogTelescopeMoveInAllow.Value;

                  
END_GET
END_PROPERTY

PROPERTY bogTurretCtClockWiseMoveAllowRawValue : BOOL
GET
                    bogTurretCtClockWiseMoveAllowRawValue := bogTurretCtClockWiseMoveAllow.Value;

                  
END_GET
END_PROPERTY

PROPERTY bogTurretClockWiseMoveAllowRawValue : BOOL
GET
                    bogTurretClockWiseMoveAllowRawValue := bogTurretClockWiseMoveAllow.Value;

                  
END_GET
END_PROPERTY

PROPERTY bogBasketRotCtClockWiseMoveAllowRawValue : BOOL
GET
                    bogBasketRotCtClockWiseMoveAllowRawValue := bogBasketRotCtClockWiseMoveAllow.Value;

                  
END_GET
END_PROPERTY

PROPERTY bogBasketRotClockWiseMoveAllowRawValue : BOOL
GET
                    bogBasketRotClockWiseMoveAllowRawValue := bogBasketRotClockWiseMoveAllow.Value;

                  
END_GET
END_PROPERTY

PROPERTY bogBasketInclinMoveUpAllowRawValue : BOOL
GET
                    bogBasketInclinMoveUpAllowRawValue := bogBasketInclinMoveUpAllow.Value;

                  
END_GET
END_PROPERTY

PROPERTY bogBasketInclinMoveDownAllowRawValue : BOOL
GET
                    bogBasketInclinMoveDownAllowRawValue := bogBasketInclinMoveDownAllow.Value;

                  
END_GET
END_PROPERTY

PROPERTY bogVehiculeDefaultRawValue : BOOL
GET
                    bogVehiculeDefaultRawValue := bogVehiculeDefault.Value;

                  
END_GET
END_PROPERTY

PROPERTY bogTelescopeOutputPossibleRawValue : BOOL
GET
                    bogTelescopeOutputPossibleRawValue := bogTelescopeOutputPossible.Value;

                  
END_GET
END_PROPERTY

PROPERTY bogTelescopeWinderFaultRawValue : BOOL
GET
                    bogTelescopeWinderFaultRawValue := bogTelescopeWinderFault.Value;

                  
END_GET
END_PROPERTY

PROPERTY bogNacellePostSelectorRawValue : BOOL
GET
                    bogNacellePostSelectorRawValue := bogNacellePostSelector.Value;

                  
END_GET
END_PROPERTY

PROPERTY bogSTOP_On_OffRawValue : BOOL
GET
                    bogSTOP_On_OffRawValue := bogSTOP_On_Off.Value;

                  
END_GET
END_PROPERTY

PROPERTY bogSafeManSystemRawValue : BOOL
GET
                    bogSafeManSystemRawValue := bogSafeManSystem.Value;

                  
END_GET
END_PROPERTY

PROPERTY bogHighSpeedAllowRawValue : BOOL
GET
                    bogHighSpeedAllowRawValue := bogHighSpeedAllow.Value;

                  
END_GET
END_PROPERTY

PROPERTY bogAutomatiqueStopRawValue : BOOL
GET
                    bogAutomatiqueStopRawValue := bogAutomatiqueStop.Value;

                  
END_GET
END_PROPERTY

PROPERTY bogLowSpeedByFaultRawValue : BOOL
GET
                    bogLowSpeedByFaultRawValue := bogLowSpeedByFault.Value;

                  
END_GET
END_PROPERTY

PROPERTY bogMeasuringMastFaultRawValue : BOOL
GET
                    bogMeasuringMastFaultRawValue := bogMeasuringMastFault.Value;

                  
END_GET
END_PROPERTY

PROPERTY bogMeasuringMatOptionRawValue : BOOL
GET
                    bogMeasuringMatOptionRawValue := bogMeasuringMatOption.Value;

                  
END_GET
END_PROPERTY

PROPERTY bogBasketAccessLockedRawValue : BOOL
GET
                    bogBasketAccessLockedRawValue := bogBasketAccessLocked.Value;

                  
END_GET
END_PROPERTY

PROPERTY bogFilterOverloadNoActiveRawValue : BOOL
GET
                    bogFilterOverloadNoActiveRawValue := bogFilterOverloadNoActive.Value;

                  
END_GET
END_PROPERTY

PROPERTY bogAnticlockwiseBasketSlewRawValue : BOOL
GET
                    bogAnticlockwiseBasketSlewRawValue := bogAnticlockwiseBasketSlew.Value;

                  
END_GET
END_PROPERTY

PROPERTY bogClockwiseBasketSlewRawValue : BOOL
GET
                    bogClockwiseBasketSlewRawValue := bogClockwiseBasketSlew.Value;

                  
END_GET
END_PROPERTY

PROPERTY bogFlashLightForcedRawValue : BOOL
GET
                    bogFlashLightForcedRawValue := bogFlashLightForced.Value;

                  
END_GET
END_PROPERTY

PROPERTY bogBasketAccessLockOptionRawValue : BOOL
GET
                    bogBasketAccessLockOptionRawValue := bogBasketAccessLockOption.Value;

                  
END_GET
END_PROPERTY

PROPERTY bogBasketLateralStopOptionRawValue : BOOL
GET
                    bogBasketLateralStopOptionRawValue := bogBasketLateralStopOption.Value;

                  
END_GET
END_PROPERTY

PROPERTY bogBasketStepClosedRawValue : BOOL
GET
                    bogBasketStepClosedRawValue := bogBasketStepClosed.Value;

                  
END_GET
END_PROPERTY

PROPERTY bogSystemFaultRawValue : BOOL
GET
                    bogSystemFaultRawValue := bogSystemFault.Value;

                  
END_GET
END_PROPERTY

PROPERTY bogTrans1PressureSensorFaultRawValue : BOOL
GET
                    bogTrans1PressureSensorFaultRawValue := bogTrans1PressureSensorFault.Value;

                  
END_GET
END_PROPERTY

PROPERTY bogTrans2PressureSensorFaultRawValue : BOOL
GET
                    bogTrans2PressureSensorFaultRawValue := bogTrans2PressureSensorFault.Value;

                  
END_GET
END_PROPERTY

PROPERTY bogOverloadSecurityRawValue : BOOL
GET
                    bogOverloadSecurityRawValue := bogOverloadSecurity.Value;

                  
END_GET
END_PROPERTY

PROPERTY bogDeltaArmJoysCenteredTelesRawValue : BOOL
GET
                    bogDeltaArmJoysCenteredTelesRawValue := bogDeltaArmJoysCenteredTeles.Value;

                  
END_GET
END_PROPERTY

PROPERTY bogArrowJoystickCenteredTurretRawValue : BOOL
GET
                    bogArrowJoystickCenteredTurretRawValue := bogArrowJoystickCenteredTurret.Value;

                  
END_GET
END_PROPERTY

PROPERTY bogDeltaArmMoveUpRawValue : BOOL
GET
                    bogDeltaArmMoveUpRawValue := bogDeltaArmMoveUp.Value;

                  
END_GET
END_PROPERTY

PROPERTY bogDeltaArmMoveDownRawValue : BOOL
GET
                    bogDeltaArmMoveDownRawValue := bogDeltaArmMoveDown.Value;

                  
END_GET
END_PROPERTY

PROPERTY bogArrowArmMoveUpRawValue : BOOL
GET
                    bogArrowArmMoveUpRawValue := bogArrowArmMoveUp.Value;

                  
END_GET
END_PROPERTY

PROPERTY bogArrowArmMoveDownRawValue : BOOL
GET
                    bogArrowArmMoveDownRawValue := bogArrowArmMoveDown.Value;

                  
END_GET
END_PROPERTY

PROPERTY bogTelescopeMoveOutRawValue : BOOL
GET
                    bogTelescopeMoveOutRawValue := bogTelescopeMoveOut.Value;

                  
END_GET
END_PROPERTY

PROPERTY bogTelescopeMoveInRawValue : BOOL
GET
                    bogTelescopeMoveInRawValue := bogTelescopeMoveIn.Value;

                  
END_GET
END_PROPERTY

PROPERTY bogTurretCounterClockWiseMoveRawValue : BOOL
GET
                    bogTurretCounterClockWiseMoveRawValue := bogTurretCounterClockWiseMove.Value;

                  
END_GET
END_PROPERTY

PROPERTY bogTurretClockWiseMoveRawValue : BOOL
GET
                    bogTurretClockWiseMoveRawValue := bogTurretClockWiseMove.Value;

                  
END_GET
END_PROPERTY

PROPERTY bogTurretEncoderFaultRawValue : BOOL
GET
                    bogTurretEncoderFaultRawValue := bogTurretEncoderFault.Value;

                  
END_GET
END_PROPERTY

PROPERTY bogGeneratorOptionRawValue : BOOL
GET
                    bogGeneratorOptionRawValue := bogGeneratorOption.Value;

                  
END_GET
END_PROPERTY

PROPERTY bogGeneratorActiveRawValue : BOOL
GET
                    bogGeneratorActiveRawValue := bogGeneratorActive.Value;

                  
END_GET
END_PROPERTY

PROPERTY bogBattery_On_OffToolValue : BOOL
GET
                    bogBattery_On_OffToolValue := bogBattery_On_Off.Value;

                  
END_GET
END_PROPERTY

PROPERTY bogPreheat_On_OffToolValue : BOOL
GET
                    bogPreheat_On_OffToolValue := bogPreheat_On_Off.Value;

                  
END_GET
END_PROPERTY

PROPERTY bogEngine_Faillure_On_OffToolValue : BOOL
GET
                    bogEngine_Faillure_On_OffToolValue := bogEngine_Faillure_On_Off.Value;

                  
END_GET
END_PROPERTY

PROPERTY bogMaintenance_On_OffToolValue : BOOL
GET
                    bogMaintenance_On_OffToolValue := bogMaintenance_On_Off.Value;

                  
END_GET
END_PROPERTY

PROPERTY bogOil_On_OFFToolValue : BOOL
GET
                    bogOil_On_OFFToolValue := bogOil_On_OFF.Value;

                  
END_GET
END_PROPERTY

PROPERTY bogDeltaArmSectorDownToolValue : BOOL
GET
                    bogDeltaArmSectorDownToolValue := bogDeltaArmSectorDown.Value;

                  
END_GET
END_PROPERTY

PROPERTY bogArrowArmSectorDownToolValue : BOOL
GET
                    bogArrowArmSectorDownToolValue := bogArrowArmSectorDown.Value;

                  
END_GET
END_PROPERTY

PROPERTY bogPendularSectorDownToolValue : BOOL
GET
                    bogPendularSectorDownToolValue := bogPendularSectorDown.Value;

                  
END_GET
END_PROPERTY

PROPERTY bogDeltaArmInCenterToolValue : BOOL
GET
                    bogDeltaArmInCenterToolValue := bogDeltaArmInCenter.Value;

                  
END_GET
END_PROPERTY

PROPERTY bogArrowArmInCenterToolValue : BOOL
GET
                    bogArrowArmInCenterToolValue := bogArrowArmInCenter.Value;

                  
END_GET
END_PROPERTY

PROPERTY bogPendularInCenterToolValue : BOOL
GET
                    bogPendularInCenterToolValue := bogPendularInCenter.Value;

                  
END_GET
END_PROPERTY

PROPERTY bogBasketRotationInCenterToolValue : BOOL
GET
                    bogBasketRotationInCenterToolValue := bogBasketRotationInCenter.Value;

                  
END_GET
END_PROPERTY

PROPERTY bogTelescopeInCenterToolValue : BOOL
GET
                    bogTelescopeInCenterToolValue := bogTelescopeInCenter.Value;

                  
END_GET
END_PROPERTY

PROPERTY bogBasketInclinaisonInCenterToolValue : BOOL
GET
                    bogBasketInclinaisonInCenterToolValue := bogBasketInclinaisonInCenter.Value;

                  
END_GET
END_PROPERTY

PROPERTY bogDeltaArmMoveUpAllowToolValue : BOOL
GET
                    bogDeltaArmMoveUpAllowToolValue := bogDeltaArmMoveUpAllow.Value;

                  
END_GET
END_PROPERTY

PROPERTY bogDeltaArmMoveDownAllowToolValue : BOOL
GET
                    bogDeltaArmMoveDownAllowToolValue := bogDeltaArmMoveDownAllow.Value;

                  
END_GET
END_PROPERTY

PROPERTY bogArrowArmMoveUpAllowToolValue : BOOL
GET
                    bogArrowArmMoveUpAllowToolValue := bogArrowArmMoveUpAllow.Value;

                  
END_GET
END_PROPERTY

PROPERTY bogArrowArmMoveDownAllowToolValue : BOOL
GET
                    bogArrowArmMoveDownAllowToolValue := bogArrowArmMoveDownAllow.Value;

                  
END_GET
END_PROPERTY

PROPERTY bogPendularMoveUpAllowToolValue : BOOL
GET
                    bogPendularMoveUpAllowToolValue := bogPendularMoveUpAllow.Value;

                  
END_GET
END_PROPERTY

PROPERTY bogPendularMoveDownAllowToolValue : BOOL
GET
                    bogPendularMoveDownAllowToolValue := bogPendularMoveDownAllow.Value;

                  
END_GET
END_PROPERTY

PROPERTY bogTelescopeMoveOutAllowToolValue : BOOL
GET
                    bogTelescopeMoveOutAllowToolValue := bogTelescopeMoveOutAllow.Value;

                  
END_GET
END_PROPERTY

PROPERTY bogTelescopeMoveInAllowToolValue : BOOL
GET
                    bogTelescopeMoveInAllowToolValue := bogTelescopeMoveInAllow.Value;

                  
END_GET
END_PROPERTY

PROPERTY bogTurretCtClockWiseMoveAllowToolValue : BOOL
GET
                    bogTurretCtClockWiseMoveAllowToolValue := bogTurretCtClockWiseMoveAllow.Value;

                  
END_GET
END_PROPERTY

PROPERTY bogTurretClockWiseMoveAllowToolValue : BOOL
GET
                    bogTurretClockWiseMoveAllowToolValue := bogTurretClockWiseMoveAllow.Value;

                  
END_GET
END_PROPERTY

PROPERTY bogBasketRotCtClockWiseMoveAllowToolValue : BOOL
GET
                    bogBasketRotCtClockWiseMoveAllowToolValue := bogBasketRotCtClockWiseMoveAllow.Value;

                  
END_GET
END_PROPERTY

PROPERTY bogBasketRotClockWiseMoveAllowToolValue : BOOL
GET
                    bogBasketRotClockWiseMoveAllowToolValue := bogBasketRotClockWiseMoveAllow.Value;

                  
END_GET
END_PROPERTY

PROPERTY bogBasketInclinMoveUpAllowToolValue : BOOL
GET
                    bogBasketInclinMoveUpAllowToolValue := bogBasketInclinMoveUpAllow.Value;

                  
END_GET
END_PROPERTY

PROPERTY bogBasketInclinMoveDownAllowToolValue : BOOL
GET
                    bogBasketInclinMoveDownAllowToolValue := bogBasketInclinMoveDownAllow.Value;

                  
END_GET
END_PROPERTY

PROPERTY bogVehiculeDefaultToolValue : BOOL
GET
                    bogVehiculeDefaultToolValue := bogVehiculeDefault.Value;

                  
END_GET
END_PROPERTY

PROPERTY bogTelescopeOutputPossibleToolValue : BOOL
GET
                    bogTelescopeOutputPossibleToolValue := bogTelescopeOutputPossible.Value;

                  
END_GET
END_PROPERTY

PROPERTY bogTelescopeWinderFaultToolValue : BOOL
GET
                    bogTelescopeWinderFaultToolValue := bogTelescopeWinderFault.Value;

                  
END_GET
END_PROPERTY

PROPERTY bogNacellePostSelectorToolValue : BOOL
GET
                    bogNacellePostSelectorToolValue := bogNacellePostSelector.Value;

                  
END_GET
END_PROPERTY

PROPERTY bogSTOP_On_OffToolValue : BOOL
GET
                    bogSTOP_On_OffToolValue := bogSTOP_On_Off.Value;

                  
END_GET
END_PROPERTY

PROPERTY bogSafeManSystemToolValue : BOOL
GET
                    bogSafeManSystemToolValue := bogSafeManSystem.Value;

                  
END_GET
END_PROPERTY

PROPERTY bogHighSpeedAllowToolValue : BOOL
GET
                    bogHighSpeedAllowToolValue := bogHighSpeedAllow.Value;

                  
END_GET
END_PROPERTY

PROPERTY bogAutomatiqueStopToolValue : BOOL
GET
                    bogAutomatiqueStopToolValue := bogAutomatiqueStop.Value;

                  
END_GET
END_PROPERTY

PROPERTY bogLowSpeedByFaultToolValue : BOOL
GET
                    bogLowSpeedByFaultToolValue := bogLowSpeedByFault.Value;

                  
END_GET
END_PROPERTY

PROPERTY bogMeasuringMastFaultToolValue : BOOL
GET
                    bogMeasuringMastFaultToolValue := bogMeasuringMastFault.Value;

                  
END_GET
END_PROPERTY

PROPERTY bogMeasuringMatOptionToolValue : BOOL
GET
                    bogMeasuringMatOptionToolValue := bogMeasuringMatOption.Value;

                  
END_GET
END_PROPERTY

PROPERTY bogBasketAccessLockedToolValue : BOOL
GET
                    bogBasketAccessLockedToolValue := bogBasketAccessLocked.Value;

                  
END_GET
END_PROPERTY

PROPERTY bogFilterOverloadNoActiveToolValue : BOOL
GET
                    bogFilterOverloadNoActiveToolValue := bogFilterOverloadNoActive.Value;

                  
END_GET
END_PROPERTY

PROPERTY bogAnticlockwiseBasketSlewToolValue : BOOL
GET
                    bogAnticlockwiseBasketSlewToolValue := bogAnticlockwiseBasketSlew.Value;

                  
END_GET
END_PROPERTY

PROPERTY bogClockwiseBasketSlewToolValue : BOOL
GET
                    bogClockwiseBasketSlewToolValue := bogClockwiseBasketSlew.Value;

                  
END_GET
END_PROPERTY

PROPERTY bogFlashLightForcedToolValue : BOOL
GET
                    bogFlashLightForcedToolValue := bogFlashLightForced.Value;

                  
END_GET
END_PROPERTY

PROPERTY bogBasketAccessLockOptionToolValue : BOOL
GET
                    bogBasketAccessLockOptionToolValue := bogBasketAccessLockOption.Value;

                  
END_GET
END_PROPERTY

PROPERTY bogBasketLateralStopOptionToolValue : BOOL
GET
                    bogBasketLateralStopOptionToolValue := bogBasketLateralStopOption.Value;

                  
END_GET
END_PROPERTY

PROPERTY bogBasketStepClosedToolValue : BOOL
GET
                    bogBasketStepClosedToolValue := bogBasketStepClosed.Value;

                  
END_GET
END_PROPERTY

PROPERTY bogSystemFaultToolValue : BOOL
GET
                    bogSystemFaultToolValue := bogSystemFault.Value;

                  
END_GET
END_PROPERTY

PROPERTY bogTrans1PressureSensorFaultToolValue : BOOL
GET
                    bogTrans1PressureSensorFaultToolValue := bogTrans1PressureSensorFault.Value;

                  
END_GET
END_PROPERTY

PROPERTY bogTrans2PressureSensorFaultToolValue : BOOL
GET
                    bogTrans2PressureSensorFaultToolValue := bogTrans2PressureSensorFault.Value;

                  
END_GET
END_PROPERTY

PROPERTY bogOverloadSecurityToolValue : BOOL
GET
                    bogOverloadSecurityToolValue := bogOverloadSecurity.Value;

                  
END_GET
END_PROPERTY

PROPERTY bogDeltaArmJoysCenteredTelesToolValue : BOOL
GET
                    bogDeltaArmJoysCenteredTelesToolValue := bogDeltaArmJoysCenteredTeles.Value;

                  
END_GET
END_PROPERTY

PROPERTY bogArrowJoystickCenteredTurretToolValue : BOOL
GET
                    bogArrowJoystickCenteredTurretToolValue := bogArrowJoystickCenteredTurret.Value;

                  
END_GET
END_PROPERTY

PROPERTY bogDeltaArmMoveUpToolValue : BOOL
GET
                    bogDeltaArmMoveUpToolValue := bogDeltaArmMoveUp.Value;

                  
END_GET
END_PROPERTY

PROPERTY bogDeltaArmMoveDownToolValue : BOOL
GET
                    bogDeltaArmMoveDownToolValue := bogDeltaArmMoveDown.Value;

                  
END_GET
END_PROPERTY

PROPERTY bogArrowArmMoveUpToolValue : BOOL
GET
                    bogArrowArmMoveUpToolValue := bogArrowArmMoveUp.Value;

                  
END_GET
END_PROPERTY

PROPERTY bogArrowArmMoveDownToolValue : BOOL
GET
                    bogArrowArmMoveDownToolValue := bogArrowArmMoveDown.Value;

                  
END_GET
END_PROPERTY

PROPERTY bogTelescopeMoveOutToolValue : BOOL
GET
                    bogTelescopeMoveOutToolValue := bogTelescopeMoveOut.Value;

                  
END_GET
END_PROPERTY

PROPERTY bogTelescopeMoveInToolValue : BOOL
GET
                    bogTelescopeMoveInToolValue := bogTelescopeMoveIn.Value;

                  
END_GET
END_PROPERTY

PROPERTY bogTurretCounterClockWiseMoveToolValue : BOOL
GET
                    bogTurretCounterClockWiseMoveToolValue := bogTurretCounterClockWiseMove.Value;

                  
END_GET
END_PROPERTY

PROPERTY bogTurretClockWiseMoveToolValue : BOOL
GET
                    bogTurretClockWiseMoveToolValue := bogTurretClockWiseMove.Value;

                  
END_GET
END_PROPERTY

PROPERTY bogTurretEncoderFaultToolValue : BOOL
GET
                    bogTurretEncoderFaultToolValue := bogTurretEncoderFault.Value;

                  
END_GET
END_PROPERTY

PROPERTY bogGeneratorOptionToolValue : BOOL
GET
                    bogGeneratorOptionToolValue := bogGeneratorOption.Value;

                  
END_GET
END_PROPERTY

PROPERTY bogGeneratorActiveToolValue : BOOL
GET
                    bogGeneratorActiveToolValue := bogGeneratorActive.Value;

                  
END_GET
END_PROPERTY

METHOD InitializeCanSignals
                  bogBattery_On_Off.AppScalingDivisor :=1;
bogBattery_On_Off.AppScalingMultiplier :=1;
bogBattery_On_Off.AppScalingOffset :=0;
bogBattery_On_Off.AppUnit :="";
bogBattery_On_Off.CanDefault :=0;
bogBattery_On_Off.CanInit :=0;
bogBattery_On_Off.CanMax :=1;
bogBattery_On_Off.CanMin :=0;
bogBattery_On_Off.CanUnit :="";
bogBattery_On_Off.Description :="Battery Status";
bogBattery_On_Off.ErrorReaction := eErrorReaction.ERSIG_DFLT;
bogBattery_On_Off.ReceiverAdress :=1;
bogBattery_On_Off.ToolScalingDivisor :=1;
bogBattery_On_Off.ToolScalingMultiplier :=1;
bogBattery_On_Off.ToolScalingOffset :=0;
bogBattery_On_Off.ToolUnit :="";

bogPreheat_On_Off.AppScalingDivisor :=1;
bogPreheat_On_Off.AppScalingMultiplier :=1;
bogPreheat_On_Off.AppScalingOffset :=0;
bogPreheat_On_Off.AppUnit :="";
bogPreheat_On_Off.CanDefault :=0;
bogPreheat_On_Off.CanInit :=0;
bogPreheat_On_Off.CanMax :=1;
bogPreheat_On_Off.CanMin :=0;
bogPreheat_On_Off.CanUnit :="";
bogPreheat_On_Off.Description :="Preheat Status";
bogPreheat_On_Off.ErrorReaction := eErrorReaction.ERSIG_DFLT;
bogPreheat_On_Off.ReceiverAdress :=1;
bogPreheat_On_Off.ToolScalingDivisor :=1;
bogPreheat_On_Off.ToolScalingMultiplier :=1;
bogPreheat_On_Off.ToolScalingOffset :=0;
bogPreheat_On_Off.ToolUnit :="";

bogEngine_Faillure_On_Off.AppScalingDivisor :=1;
bogEngine_Faillure_On_Off.AppScalingMultiplier :=1;
bogEngine_Faillure_On_Off.AppScalingOffset :=0;
bogEngine_Faillure_On_Off.AppUnit :="";
bogEngine_Faillure_On_Off.CanDefault :=0;
bogEngine_Faillure_On_Off.CanInit :=0;
bogEngine_Faillure_On_Off.CanMax :=1;
bogEngine_Faillure_On_Off.CanMin :=0;
bogEngine_Faillure_On_Off.CanUnit :="";
bogEngine_Faillure_On_Off.Description :="Engine Faillure Status";
bogEngine_Faillure_On_Off.ErrorReaction := eErrorReaction.ERSIG_DFLT;
bogEngine_Faillure_On_Off.ReceiverAdress :=1;
bogEngine_Faillure_On_Off.ToolScalingDivisor :=1;
bogEngine_Faillure_On_Off.ToolScalingMultiplier :=1;
bogEngine_Faillure_On_Off.ToolScalingOffset :=0;
bogEngine_Faillure_On_Off.ToolUnit :="";

bogMaintenance_On_Off.AppScalingDivisor :=1;
bogMaintenance_On_Off.AppScalingMultiplier :=1;
bogMaintenance_On_Off.AppScalingOffset :=0;
bogMaintenance_On_Off.AppUnit :="";
bogMaintenance_On_Off.CanDefault :=0;
bogMaintenance_On_Off.CanInit :=0;
bogMaintenance_On_Off.CanMax :=1;
bogMaintenance_On_Off.CanMin :=0;
bogMaintenance_On_Off.CanUnit :="";
bogMaintenance_On_Off.Description :="Maintenance Status";
bogMaintenance_On_Off.ErrorReaction := eErrorReaction.ERSIG_DFLT;
bogMaintenance_On_Off.ReceiverAdress :=1;
bogMaintenance_On_Off.ToolScalingDivisor :=1;
bogMaintenance_On_Off.ToolScalingMultiplier :=1;
bogMaintenance_On_Off.ToolScalingOffset :=0;
bogMaintenance_On_Off.ToolUnit :="";

bogOil_On_OFF.AppScalingDivisor :=1;
bogOil_On_OFF.AppScalingMultiplier :=1;
bogOil_On_OFF.AppScalingOffset :=0;
bogOil_On_OFF.AppUnit :="";
bogOil_On_OFF.CanDefault :=0;
bogOil_On_OFF.CanInit :=0;
bogOil_On_OFF.CanMax :=1;
bogOil_On_OFF.CanMin :=0;
bogOil_On_OFF.CanUnit :="";
bogOil_On_OFF.Description :="Oil Status";
bogOil_On_OFF.ErrorReaction := eErrorReaction.ERSIG_DFLT;
bogOil_On_OFF.ReceiverAdress :=1;
bogOil_On_OFF.ToolScalingDivisor :=1;
bogOil_On_OFF.ToolScalingMultiplier :=1;
bogOil_On_OFF.ToolScalingOffset :=0;
bogOil_On_OFF.ToolUnit :="";

bogDeltaArmSectorDown.AppScalingDivisor :=1;
bogDeltaArmSectorDown.AppScalingMultiplier :=1;
bogDeltaArmSectorDown.AppScalingOffset :=0;
bogDeltaArmSectorDown.AppUnit :="";
bogDeltaArmSectorDown.CanDefault :=0;
bogDeltaArmSectorDown.CanInit :=0;
bogDeltaArmSectorDown.CanMax :=1;
bogDeltaArmSectorDown.CanMin :=0;
bogDeltaArmSectorDown.CanUnit :="";
bogDeltaArmSectorDown.Description :="Delta Arm Sector Down";
bogDeltaArmSectorDown.ErrorReaction := eErrorReaction.ERSIG_DFLT;
bogDeltaArmSectorDown.ReceiverAdress :=1;
bogDeltaArmSectorDown.ToolScalingDivisor :=1;
bogDeltaArmSectorDown.ToolScalingMultiplier :=1;
bogDeltaArmSectorDown.ToolScalingOffset :=0;
bogDeltaArmSectorDown.ToolUnit :="";

bogArrowArmSectorDown.AppScalingDivisor :=1;
bogArrowArmSectorDown.AppScalingMultiplier :=1;
bogArrowArmSectorDown.AppScalingOffset :=0;
bogArrowArmSectorDown.AppUnit :="";
bogArrowArmSectorDown.CanDefault :=0;
bogArrowArmSectorDown.CanInit :=0;
bogArrowArmSectorDown.CanMax :=1;
bogArrowArmSectorDown.CanMin :=0;
bogArrowArmSectorDown.CanUnit :="";
bogArrowArmSectorDown.Description :="Arrow Arm Sector Down";
bogArrowArmSectorDown.ErrorReaction := eErrorReaction.ERSIG_DFLT;
bogArrowArmSectorDown.ReceiverAdress :=1;
bogArrowArmSectorDown.ToolScalingDivisor :=1;
bogArrowArmSectorDown.ToolScalingMultiplier :=1;
bogArrowArmSectorDown.ToolScalingOffset :=0;
bogArrowArmSectorDown.ToolUnit :="";

bogPendularSectorDown.AppScalingDivisor :=1;
bogPendularSectorDown.AppScalingMultiplier :=1;
bogPendularSectorDown.AppScalingOffset :=0;
bogPendularSectorDown.AppUnit :="";
bogPendularSectorDown.CanDefault :=0;
bogPendularSectorDown.CanInit :=0;
bogPendularSectorDown.CanMax :=1;
bogPendularSectorDown.CanMin :=0;
bogPendularSectorDown.CanUnit :="";
bogPendularSectorDown.Description :="Pendular Sector Down";
bogPendularSectorDown.ErrorReaction := eErrorReaction.ERSIG_DFLT;
bogPendularSectorDown.ReceiverAdress :=1;
bogPendularSectorDown.ToolScalingDivisor :=1;
bogPendularSectorDown.ToolScalingMultiplier :=1;
bogPendularSectorDown.ToolScalingOffset :=0;
bogPendularSectorDown.ToolUnit :="";

bogDeltaArmInCenter.AppScalingDivisor :=1;
bogDeltaArmInCenter.AppScalingMultiplier :=1;
bogDeltaArmInCenter.AppScalingOffset :=0;
bogDeltaArmInCenter.AppUnit :="";
bogDeltaArmInCenter.CanDefault :=0;
bogDeltaArmInCenter.CanInit :=0;
bogDeltaArmInCenter.CanMax :=1;
bogDeltaArmInCenter.CanMin :=0;
bogDeltaArmInCenter.CanUnit :="";
bogDeltaArmInCenter.Description :="Delta Arm in Center";
bogDeltaArmInCenter.ErrorReaction := eErrorReaction.ERSIG_DFLT;
bogDeltaArmInCenter.ReceiverAdress :=1;
bogDeltaArmInCenter.ToolScalingDivisor :=1;
bogDeltaArmInCenter.ToolScalingMultiplier :=1;
bogDeltaArmInCenter.ToolScalingOffset :=0;
bogDeltaArmInCenter.ToolUnit :="";

bogArrowArmInCenter.AppScalingDivisor :=1;
bogArrowArmInCenter.AppScalingMultiplier :=1;
bogArrowArmInCenter.AppScalingOffset :=0;
bogArrowArmInCenter.AppUnit :="";
bogArrowArmInCenter.CanDefault :=0;
bogArrowArmInCenter.CanInit :=0;
bogArrowArmInCenter.CanMax :=1;
bogArrowArmInCenter.CanMin :=0;
bogArrowArmInCenter.CanUnit :="";
bogArrowArmInCenter.Description :="Arrow Arm in Center";
bogArrowArmInCenter.ErrorReaction := eErrorReaction.ERSIG_DFLT;
bogArrowArmInCenter.ReceiverAdress :=1;
bogArrowArmInCenter.ToolScalingDivisor :=1;
bogArrowArmInCenter.ToolScalingMultiplier :=1;
bogArrowArmInCenter.ToolScalingOffset :=0;
bogArrowArmInCenter.ToolUnit :="";

bogPendularInCenter.AppScalingDivisor :=1;
bogPendularInCenter.AppScalingMultiplier :=1;
bogPendularInCenter.AppScalingOffset :=0;
bogPendularInCenter.AppUnit :="";
bogPendularInCenter.CanDefault :=0;
bogPendularInCenter.CanInit :=0;
bogPendularInCenter.CanMax :=1;
bogPendularInCenter.CanMin :=0;
bogPendularInCenter.CanUnit :="";
bogPendularInCenter.Description :="Pendular in Center";
bogPendularInCenter.ErrorReaction := eErrorReaction.ERSIG_DFLT;
bogPendularInCenter.ReceiverAdress :=1;
bogPendularInCenter.ToolScalingDivisor :=1;
bogPendularInCenter.ToolScalingMultiplier :=1;
bogPendularInCenter.ToolScalingOffset :=0;
bogPendularInCenter.ToolUnit :="";

bogBasketRotationInCenter.AppScalingDivisor :=1;
bogBasketRotationInCenter.AppScalingMultiplier :=1;
bogBasketRotationInCenter.AppScalingOffset :=0;
bogBasketRotationInCenter.AppUnit :="";
bogBasketRotationInCenter.CanDefault :=0;
bogBasketRotationInCenter.CanInit :=0;
bogBasketRotationInCenter.CanMax :=1;
bogBasketRotationInCenter.CanMin :=0;
bogBasketRotationInCenter.CanUnit :="";
bogBasketRotationInCenter.Description :="Basket Rotation in Center";
bogBasketRotationInCenter.ErrorReaction := eErrorReaction.ERSIG_DFLT;
bogBasketRotationInCenter.ReceiverAdress :=1;
bogBasketRotationInCenter.ToolScalingDivisor :=1;
bogBasketRotationInCenter.ToolScalingMultiplier :=1;
bogBasketRotationInCenter.ToolScalingOffset :=0;
bogBasketRotationInCenter.ToolUnit :="";

bogTelescopeInCenter.AppScalingDivisor :=1;
bogTelescopeInCenter.AppScalingMultiplier :=1;
bogTelescopeInCenter.AppScalingOffset :=0;
bogTelescopeInCenter.AppUnit :="";
bogTelescopeInCenter.CanDefault :=0;
bogTelescopeInCenter.CanInit :=0;
bogTelescopeInCenter.CanMax :=1;
bogTelescopeInCenter.CanMin :=0;
bogTelescopeInCenter.CanUnit :="";
bogTelescopeInCenter.Description :="Telescope in Center";
bogTelescopeInCenter.ErrorReaction := eErrorReaction.ERSIG_DFLT;
bogTelescopeInCenter.ReceiverAdress :=1;
bogTelescopeInCenter.ToolScalingDivisor :=1;
bogTelescopeInCenter.ToolScalingMultiplier :=1;
bogTelescopeInCenter.ToolScalingOffset :=0;
bogTelescopeInCenter.ToolUnit :="";

bogBasketInclinaisonInCenter.AppScalingDivisor :=1;
bogBasketInclinaisonInCenter.AppScalingMultiplier :=1;
bogBasketInclinaisonInCenter.AppScalingOffset :=0;
bogBasketInclinaisonInCenter.AppUnit :="";
bogBasketInclinaisonInCenter.CanDefault :=0;
bogBasketInclinaisonInCenter.CanInit :=0;
bogBasketInclinaisonInCenter.CanMax :=1;
bogBasketInclinaisonInCenter.CanMin :=0;
bogBasketInclinaisonInCenter.CanUnit :="";
bogBasketInclinaisonInCenter.Description :="Basket Inclinaison in Center";
bogBasketInclinaisonInCenter.ErrorReaction := eErrorReaction.ERSIG_DFLT;
bogBasketInclinaisonInCenter.ReceiverAdress :=1;
bogBasketInclinaisonInCenter.ToolScalingDivisor :=1;
bogBasketInclinaisonInCenter.ToolScalingMultiplier :=1;
bogBasketInclinaisonInCenter.ToolScalingOffset :=0;
bogBasketInclinaisonInCenter.ToolUnit :="";

bogDeltaArmMoveUpAllow.AppScalingDivisor :=1;
bogDeltaArmMoveUpAllow.AppScalingMultiplier :=1;
bogDeltaArmMoveUpAllow.AppScalingOffset :=0;
bogDeltaArmMoveUpAllow.AppUnit :="";
bogDeltaArmMoveUpAllow.CanDefault :=0;
bogDeltaArmMoveUpAllow.CanInit :=0;
bogDeltaArmMoveUpAllow.CanMax :=1;
bogDeltaArmMoveUpAllow.CanMin :=0;
bogDeltaArmMoveUpAllow.CanUnit :="";
bogDeltaArmMoveUpAllow.Description :="Delta Arm Move Up Allowed";
bogDeltaArmMoveUpAllow.ErrorReaction := eErrorReaction.ERSIG_DFLT;
bogDeltaArmMoveUpAllow.ReceiverAdress :=1;
bogDeltaArmMoveUpAllow.ToolScalingDivisor :=1;
bogDeltaArmMoveUpAllow.ToolScalingMultiplier :=1;
bogDeltaArmMoveUpAllow.ToolScalingOffset :=0;
bogDeltaArmMoveUpAllow.ToolUnit :="";

bogDeltaArmMoveDownAllow.AppScalingDivisor :=1;
bogDeltaArmMoveDownAllow.AppScalingMultiplier :=1;
bogDeltaArmMoveDownAllow.AppScalingOffset :=0;
bogDeltaArmMoveDownAllow.AppUnit :="";
bogDeltaArmMoveDownAllow.CanDefault :=0;
bogDeltaArmMoveDownAllow.CanInit :=0;
bogDeltaArmMoveDownAllow.CanMax :=1;
bogDeltaArmMoveDownAllow.CanMin :=0;
bogDeltaArmMoveDownAllow.CanUnit :="";
bogDeltaArmMoveDownAllow.Description :="Delta Arm Move Down Allowed";
bogDeltaArmMoveDownAllow.ErrorReaction := eErrorReaction.ERSIG_DFLT;
bogDeltaArmMoveDownAllow.ReceiverAdress :=1;
bogDeltaArmMoveDownAllow.ToolScalingDivisor :=1;
bogDeltaArmMoveDownAllow.ToolScalingMultiplier :=1;
bogDeltaArmMoveDownAllow.ToolScalingOffset :=0;
bogDeltaArmMoveDownAllow.ToolUnit :="";

bogArrowArmMoveUpAllow.AppScalingDivisor :=1;
bogArrowArmMoveUpAllow.AppScalingMultiplier :=1;
bogArrowArmMoveUpAllow.AppScalingOffset :=0;
bogArrowArmMoveUpAllow.AppUnit :="";
bogArrowArmMoveUpAllow.CanDefault :=0;
bogArrowArmMoveUpAllow.CanInit :=0;
bogArrowArmMoveUpAllow.CanMax :=1;
bogArrowArmMoveUpAllow.CanMin :=0;
bogArrowArmMoveUpAllow.CanUnit :="";
bogArrowArmMoveUpAllow.Description :="Arrow Arm Move Up Allowed";
bogArrowArmMoveUpAllow.ErrorReaction := eErrorReaction.ERSIG_DFLT;
bogArrowArmMoveUpAllow.ReceiverAdress :=1;
bogArrowArmMoveUpAllow.ToolScalingDivisor :=1;
bogArrowArmMoveUpAllow.ToolScalingMultiplier :=1;
bogArrowArmMoveUpAllow.ToolScalingOffset :=0;
bogArrowArmMoveUpAllow.ToolUnit :="";

bogArrowArmMoveDownAllow.AppScalingDivisor :=1;
bogArrowArmMoveDownAllow.AppScalingMultiplier :=1;
bogArrowArmMoveDownAllow.AppScalingOffset :=0;
bogArrowArmMoveDownAllow.AppUnit :="";
bogArrowArmMoveDownAllow.CanDefault :=0;
bogArrowArmMoveDownAllow.CanInit :=0;
bogArrowArmMoveDownAllow.CanMax :=1;
bogArrowArmMoveDownAllow.CanMin :=0;
bogArrowArmMoveDownAllow.CanUnit :="";
bogArrowArmMoveDownAllow.Description :="Arrow Arm Move Down Allowed";
bogArrowArmMoveDownAllow.ErrorReaction := eErrorReaction.ERSIG_DFLT;
bogArrowArmMoveDownAllow.ReceiverAdress :=1;
bogArrowArmMoveDownAllow.ToolScalingDivisor :=1;
bogArrowArmMoveDownAllow.ToolScalingMultiplier :=1;
bogArrowArmMoveDownAllow.ToolScalingOffset :=0;
bogArrowArmMoveDownAllow.ToolUnit :="";

bogPendularMoveUpAllow.AppScalingDivisor :=1;
bogPendularMoveUpAllow.AppScalingMultiplier :=1;
bogPendularMoveUpAllow.AppScalingOffset :=0;
bogPendularMoveUpAllow.AppUnit :="";
bogPendularMoveUpAllow.CanDefault :=0;
bogPendularMoveUpAllow.CanInit :=0;
bogPendularMoveUpAllow.CanMax :=1;
bogPendularMoveUpAllow.CanMin :=0;
bogPendularMoveUpAllow.CanUnit :="";
bogPendularMoveUpAllow.Description :="Pendular Move Up Allowed";
bogPendularMoveUpAllow.ErrorReaction := eErrorReaction.ERSIG_DFLT;
bogPendularMoveUpAllow.ReceiverAdress :=1;
bogPendularMoveUpAllow.ToolScalingDivisor :=1;
bogPendularMoveUpAllow.ToolScalingMultiplier :=1;
bogPendularMoveUpAllow.ToolScalingOffset :=0;
bogPendularMoveUpAllow.ToolUnit :="";

bogPendularMoveDownAllow.AppScalingDivisor :=1;
bogPendularMoveDownAllow.AppScalingMultiplier :=1;
bogPendularMoveDownAllow.AppScalingOffset :=0;
bogPendularMoveDownAllow.AppUnit :="";
bogPendularMoveDownAllow.CanDefault :=0;
bogPendularMoveDownAllow.CanInit :=0;
bogPendularMoveDownAllow.CanMax :=1;
bogPendularMoveDownAllow.CanMin :=0;
bogPendularMoveDownAllow.CanUnit :="";
bogPendularMoveDownAllow.Description :="Pendular Move Down Allowed";
bogPendularMoveDownAllow.ErrorReaction := eErrorReaction.ERSIG_DFLT;
bogPendularMoveDownAllow.ReceiverAdress :=1;
bogPendularMoveDownAllow.ToolScalingDivisor :=1;
bogPendularMoveDownAllow.ToolScalingMultiplier :=1;
bogPendularMoveDownAllow.ToolScalingOffset :=0;
bogPendularMoveDownAllow.ToolUnit :="";

bogTelescopeMoveOutAllow.AppScalingDivisor :=1;
bogTelescopeMoveOutAllow.AppScalingMultiplier :=1;
bogTelescopeMoveOutAllow.AppScalingOffset :=0;
bogTelescopeMoveOutAllow.AppUnit :="";
bogTelescopeMoveOutAllow.CanDefault :=0;
bogTelescopeMoveOutAllow.CanInit :=0;
bogTelescopeMoveOutAllow.CanMax :=1;
bogTelescopeMoveOutAllow.CanMin :=0;
bogTelescopeMoveOutAllow.CanUnit :="";
bogTelescopeMoveOutAllow.Description :="Telescope Move Out Allowed";
bogTelescopeMoveOutAllow.ErrorReaction := eErrorReaction.ERSIG_DFLT;
bogTelescopeMoveOutAllow.ReceiverAdress :=1;
bogTelescopeMoveOutAllow.ToolScalingDivisor :=1;
bogTelescopeMoveOutAllow.ToolScalingMultiplier :=1;
bogTelescopeMoveOutAllow.ToolScalingOffset :=0;
bogTelescopeMoveOutAllow.ToolUnit :="";

bogTelescopeMoveInAllow.AppScalingDivisor :=1;
bogTelescopeMoveInAllow.AppScalingMultiplier :=1;
bogTelescopeMoveInAllow.AppScalingOffset :=0;
bogTelescopeMoveInAllow.AppUnit :="";
bogTelescopeMoveInAllow.CanDefault :=0;
bogTelescopeMoveInAllow.CanInit :=0;
bogTelescopeMoveInAllow.CanMax :=1;
bogTelescopeMoveInAllow.CanMin :=0;
bogTelescopeMoveInAllow.CanUnit :="";
bogTelescopeMoveInAllow.Description :="Telescope Move In Allowed";
bogTelescopeMoveInAllow.ErrorReaction := eErrorReaction.ERSIG_DFLT;
bogTelescopeMoveInAllow.ReceiverAdress :=1;
bogTelescopeMoveInAllow.ToolScalingDivisor :=1;
bogTelescopeMoveInAllow.ToolScalingMultiplier :=1;
bogTelescopeMoveInAllow.ToolScalingOffset :=0;
bogTelescopeMoveInAllow.ToolUnit :="";

bogTurretCtClockWiseMoveAllow.AppScalingDivisor :=1;
bogTurretCtClockWiseMoveAllow.AppScalingMultiplier :=1;
bogTurretCtClockWiseMoveAllow.AppScalingOffset :=0;
bogTurretCtClockWiseMoveAllow.AppUnit :="";
bogTurretCtClockWiseMoveAllow.CanDefault :=0;
bogTurretCtClockWiseMoveAllow.CanInit :=0;
bogTurretCtClockWiseMoveAllow.CanMax :=1;
bogTurretCtClockWiseMoveAllow.CanMin :=0;
bogTurretCtClockWiseMoveAllow.CanUnit :="";
bogTurretCtClockWiseMoveAllow.Description :="Turret Counter Clockwise Move Allowed";
bogTurretCtClockWiseMoveAllow.ErrorReaction := eErrorReaction.ERSIG_DFLT;
bogTurretCtClockWiseMoveAllow.ReceiverAdress :=1;
bogTurretCtClockWiseMoveAllow.ToolScalingDivisor :=1;
bogTurretCtClockWiseMoveAllow.ToolScalingMultiplier :=1;
bogTurretCtClockWiseMoveAllow.ToolScalingOffset :=0;
bogTurretCtClockWiseMoveAllow.ToolUnit :="";

bogTurretClockWiseMoveAllow.AppScalingDivisor :=1;
bogTurretClockWiseMoveAllow.AppScalingMultiplier :=1;
bogTurretClockWiseMoveAllow.AppScalingOffset :=0;
bogTurretClockWiseMoveAllow.AppUnit :="";
bogTurretClockWiseMoveAllow.CanDefault :=0;
bogTurretClockWiseMoveAllow.CanInit :=0;
bogTurretClockWiseMoveAllow.CanMax :=1;
bogTurretClockWiseMoveAllow.CanMin :=0;
bogTurretClockWiseMoveAllow.CanUnit :="";
bogTurretClockWiseMoveAllow.Description :="Turret Clockwise Move Allowed";
bogTurretClockWiseMoveAllow.ErrorReaction := eErrorReaction.ERSIG_DFLT;
bogTurretClockWiseMoveAllow.ReceiverAdress :=1;
bogTurretClockWiseMoveAllow.ToolScalingDivisor :=1;
bogTurretClockWiseMoveAllow.ToolScalingMultiplier :=1;
bogTurretClockWiseMoveAllow.ToolScalingOffset :=0;
bogTurretClockWiseMoveAllow.ToolUnit :="";

